LIN {X 0,Y 388.973,Z 474.655,A -85,B 0,C 180,E1 -11902.254,E2 -11902.254} C_VEL
LIN {X 0,Y 390.4,Z 456.308,A -85,B 0,C 180,E1 -11905.598,E2 -11905.598} C_VEL
LIN {X 0,Y 390.366,Z 451.941,A -85,B 0,C 180,E1 -11906.461,E2 -11906.461} C_VEL
LIN {X 0,Y 388.692,Z 443.592,A -85,B 0,C 180,E1 -11908.299,E2 -11908.299} C_VEL
LIN {X 0,Y 386.693,Z 436.556,A -85,B 0,C 180,E1 -11909.986,E2 -11909.986} C_VEL
LIN {X 0,Y 383.976,Z 428.562,A -85,B 0,C 180,E1 -11912.059,E2 -11912.059} C_VEL
LIN {X 0,Y 383.014,Z 425.779,A -85,B 0,C 180,E1 -11912.861,E2 -11912.861} C_VEL
LIN {X 0,Y 383.034,Z 425.772,A -85,B 0,C 180,E1 -11916.164,E2 -11916.164} C_VEL
LIN {X 0,Y 383.01,Z 425.774,A -85,B 0,C 180,E1 -11919.958,E2 -11919.958} C_VEL
LIN {X 0,Y 383.007,Z 425.776,A -85,B 0,C 180,E1 -11922.779,E2 -11922.779} C_VEL
LIN {X 0,Y 382.999,Z 425.778,A -85,B 0,C 180,E1 -11925.789,E2 -11925.789} C_VEL
LIN {X 0,Y 382.99,Z 425.776,A -85,B 0,C 180,E1 -11928.796,E2 -11928.796} C_VEL
LIN {X 0,Y 383.001,Z 425.776,A -85,B 0,C 180,E1 -11932.096,E2 -11932.096} C_VEL
LIN {X 0,Y 383.02,Z 425.775,A -85,B 0,C 180,E1 -11935.332,E2 -11935.332} C_VEL
LIN {X 0,Y 383.022,Z 425.882,A -85,B 0,C 180,E1 -11938.509,E2 -11938.509} C_VEL
LIN {X 0,Y 386.811,Z 443.638,A -85,B 0,C 180,E1 -11942.071,E2 -11942.071} C_VEL
LIN {X 0,Y 387.334,Z 447.211,A -85,B 0,C 180,E1 -11942.759,E2 -11942.759} C_VEL
LIN {X 0,Y 386.152,Z 463.005,A -85,B 0,C 180,E1 -11945.62,E2 -11945.62} C_VEL
LIN {X 0,Y 385.72,Z 469.471,A -85,B 0,C 180,E1 -11946.76,E2 -11946.76} C_VEL
LIN {X 0,Y 387.23,Z 483.824,A -85,B 0,C 180,E1 -11947.858,E2 -11947.858} C_VEL
LIN {X 0,Y 389.694,Z 500.187,A -85,B 0,C 180,E1 -11948.651,E2 -11948.651} C_VEL
LIN {X 0,Y 391.644,Z 523.161,A -85,B 0,C 180,E1 -11949.556,E2 -11949.556} C_VEL
LIN {X 0,Y 388.702,Z 598.961,A -85,B 0,C 180,E1 -11951.588,E2 -11951.588} C_VEL
LIN {X 0,Y 388.096,Z 612.843,A -85,B 0,C 180,E1 -11952.036,E2 -11952.036} C_VEL
LIN {X 0,Y 387.433,Z 625.993,A -85,B 0,C 180,E1 -11952.652,E2 -11952.652} C_VEL
LIN {X 0,Y 386.462,Z 638.87,A -85,B 0,C 180,E1 -11953.492,E2 -11953.492} C_VEL
LIN {X 0,Y 385.655,Z 649.554,A -85,B 0,C 180,E1 -11954.407,E2 -11954.407} C_VEL
LIN {X 0,Y 384.808,Z 660.326,A -85,B 0,C 180,E1 -11955.578,E2 -11955.578} C_VEL
LIN {X 0,Y 383.983,Z 669.284,A -85,B 0,C 180,E1 -11956.774,E2 -11956.774} C_VEL
LIN {X 0,Y 383.117,Z 678.923,A -85,B 0,C 180,E1 -11958.358,E2 -11958.358} C_VEL
LIN {X 0,Y 382.509,Z 686.731,A -85,B 0,C 180,E1 -11959.948,E2 -11959.948} C_VEL
LIN {X 0,Y 382.085,Z 692.947,A -85,B 0,C 180,E1 -11961.538,E2 -11961.538} C_VEL
LIN {X 0,Y 381.834,Z 697.818,A -85,B 0,C 180,E1 -11963.129,E2 -11963.129} C_VEL
LIN {X 0,Y 381.699,Z 701.49,A -85,B 0,C 180,E1 -11964.718,E2 -11964.718} C_VEL
LIN {X 0,Y 381.686,Z 703.304,A -85,B 0,C 180,E1 -11965.776,E2 -11965.776} C_VEL
LIN {X 0,Y 381.62,Z 704.68,A -85,B 0,C 180,E1 -11966.833,E2 -11966.833} C_VEL
LIN {X 0,Y 381.631,Z 705.587,A -85,B 0,C 180,E1 -11967.889,E2 -11967.889} C_VEL
LIN {X 0,Y 381.687,Z 706.203,A -85,B 0,C 180,E1 -11970,E2 -11970} C_VEL
LIN {X 0,Y 381.677,Z 705.98,A -85,B 0,C 180,E1 -11971.055,E2 -11971.055} C_VEL
LIN {X 0,Y 381.636,Z 705.361,A -85,B 0,C 180,E1 -11972.111,E2 -11972.111} C_VEL
LIN {X 0,Y 381.625,Z 704.35,A -85,B 0,C 180,E1 -11973.167,E2 -11973.167} C_VEL
LIN {X 0,Y 381.69,Z 702.918,A -85,B 0,C 180,E1 -11974.224,E2 -11974.224} C_VEL
LIN {X 0,Y 381.756,Z 698.991,A -85,B 0,C 180,E1 -11976.213,E2 -11976.213} C_VEL
LIN {X 0,Y 381.995,Z 694.268,A -85,B 0,C 180,E1 -11977.931,E2 -11977.931} C_VEL
LIN {X 0,Y 382.45,Z 687.532,A -85,B 0,C 180,E1 -11979.787,E2 -11979.787} C_VEL
LIN {X 0,Y 383.006,Z 680.171,A -85,B 0,C 180,E1 -11981.377,E2 -11981.377} C_VEL
LIN {X 0,Y 383.706,Z 672.652,A -85,B 0,C 180,E1 -11982.697,E2 -11982.697} C_VEL
LIN {X 0,Y 384.542,Z 663.035,A -85,B 0,C 180,E1 -11984.079,E2 -11984.079} C_VEL
LIN {X 0,Y 385.394,Z 652.076,A -85,B 0,C 180,E1 -11985.333,E2 -11985.333} C_VEL
LIN {X 0,Y 386.372,Z 640.484,A -85,B 0,C 180,E1 -11986.376,E2 -11986.376} C_VEL
LIN {X 0,Y 387.296,Z 628.071,A -85,B 0,C 180,E1 -11987.218,E2 -11987.218} C_VEL
LIN {X 0,Y 388.001,Z 614.983,A -85,B 0,C 180,E1 -11987.866,E2 -11987.866} C_VEL
LIN {X 0,Y 389.326,Z 594.994,A -85,B 0,C 180,E1 -11988.722,E2 -11988.722} C_VEL
LIN {X 0,Y 390.088,Z 575.45,A -85,B 0,C 180,E1 -11989.264,E2 -11989.264} C_VEL
LIN {X 0,Y 391.896,Z 521.918,A -85,B 0,C 180,E1 -11990.668,E2 -11990.668} C_VEL
LIN {X 0,Y 390.385,Z 503.692,A -85,B 0,C 180,E1 -11991.348,E2 -11991.348} C_VEL
LIN {X 0,Y 387.383,Z 484.338,A -85,B 0,C 180,E1 -11992.23,E2 -11992.23} C_VEL
LIN {X 0,Y 386.082,Z 477.709,A -85,B 0,C 180,E1 -11992.58,E2 -11992.58} C_VEL
LIN {X 0,Y 387.967,Z 460.117,A -85,B 0,C 180,E1 -11996.059,E2 -11996.059} C_VEL
LIN {X 0,Y 389.025,Z 450.691,A -85,B 0,C 180,E1 -11998.015,E2 -11998.015} C_VEL
LIN {X 0,Y 387.628,Z 442.996,A -85,B 0,C 180,E1 -11999.932,E2 -11999.932} C_VEL
LIN {X 0,Y 385.295,Z 433.56,A -85,B 0,C 180,E1 -12002.584,E2 -12002.584} C_VEL
LIN {X 0,Y 383.068,Z 425.77,A -85,B 0,C 180,E1 -12005.144,E2 -12005.144} C_VEL
LIN {X 0,Y 383.003,Z 425.777,A -85,B 0,C 180,E1 -12008.601,E2 -12008.601} C_VEL
LIN {X 0,Y 382.983,Z 425.78,A -85,B 0,C 180,E1 -12011.348,E2 -12011.348} C_VEL
LIN {X 0,Y 382.997,Z 425.778,A -85,B 0,C 180,E1 -12014.303,E2 -12014.303} C_VEL
LIN {X 0,Y 383.012,Z 425.777,A -85,B 0,C 180,E1 -12017.24,E2 -12017.24} C_VEL
LIN {X 0,Y 383.017,Z 425.775,A -85,B 0,C 180,E1 -12020.413,E2 -12020.413} C_VEL
LIN {X 0,Y 383.027,Z 425.772,A -85,B 0,C 180,E1 -12024.045,E2 -12024.045} C_VEL
LIN {X 0,Y 382.989,Z 425.778,A -85,B 0,C 180,E1 -12027.578,E2 -12027.578} C_VEL
LIN {X 0,Y 382.994,Z 425.778,A -85,B 0,C 180,E1 -12030.3,E2 -12030.3} C_VEL
LIN {X 0,Y 383.082,Z 425.769,A -85,B 0,C 180,E1 -12034.021,E2 -12034.021} C_VEL
LIN {X 0,Y 383.06,Z 425.881,A -85,B 0,C 180,E1 -12037.093,E2 -12037.093} C_VEL
LIN {X 0,Y 383.156,Z 426.461,A -85,B 0,C 180,E1 -12037.246,E2 -12037.246} C_VEL
LIN {X 0,Y 384.382,Z 429.177,A -85,B 0,C 180,E1 -12037.475,E2 -12037.475} C_VEL
LIN {X 0,Y 385.896,Z 431.761,A -85,B 0,C 180,E1 -12037.727,E2 -12037.727} C_VEL
LIN {X 0,Y 391.372,Z 442.113,A -85,B 0,C 180,E1 -12038.631,E2 -12038.631} C_VEL
LIN {X 0,Y 394.03,Z 448.2,A -85,B 0,C 180,E1 -12039.076,E2 -12039.076} C_VEL
LIN {X 0,Y 391.15,Z 515.753,A -85,B 0,C 180,E1 -12040.892,E2 -12040.892} C_VEL
LIN {X 0,Y 390.648,Z 532.946,A -85,B 0,C 180,E1 -12041.411,E2 -12041.411} C_VEL
LIN {X 0,Y 390.136,Z 545.919,A -85,B 0,C 180,E1 -12042.031,E2 -12042.031} C_VEL
LIN {X 0,Y 389.456,Z 558.538,A -85,B 0,C 180,E1 -12042.853,E2 -12042.853} C_VEL
LIN {X 0,Y 388.498,Z 570.752,A -85,B 0,C 180,E1 -12043.891,E2 -12043.891} C_VEL
LIN {X 0,Y 387.531,Z 581.387,A -85,B 0,C 180,E1 -12045.023,E2 -12045.023} C_VEL
LIN {X 0,Y 386.635,Z 591.162,A -85,B 0,C 180,E1 -12046.331,E2 -12046.331} C_VEL
LIN {X 0,Y 385.652,Z 600.607,A -85,B 0,C 180,E1 -12047.903,E2 -12047.903} C_VEL
LIN {X 0,Y 384.683,Z 608.126,A -85,B 0,C 180,E1 -12049.473,E2 -12049.473} C_VEL
LIN {X 0,Y 383.999,Z 614.699,A -85,B 0,C 180,E1 -12051.235,E2 -12051.235} C_VEL
LIN {X 0,Y 383.308,Z 618.819,A -85,B 0,C 180,E1 -12052.626,E2 -12052.626} C_VEL
LIN {X 0,Y 383.106,Z 621.312,A -85,B 0,C 180,E1 -12053.681,E2 -12053.681} C_VEL
LIN {X 0,Y 382.945,Z 623.281,A -85,B 0,C 180,E1 -12054.735,E2 -12054.735} C_VEL
LIN {X 0,Y 382.672,Z 624.822,A -85,B 0,C 180,E1 -12055.787,E2 -12055.787} C_VEL
LIN {X 0,Y 382.364,Z 625.951,A -85,B 0,C 180,E1 -12056.839,E2 -12056.839} C_VEL
LIN {X 0,Y 382.146,Z 626.62,A -85,B 0,C 180,E1 -12057.892,E2 -12057.892} C_VEL
LIN {X 0,Y 382.038,Z 626.843,A -85,B 0,C 180,E1 -12058.946,E2 -12058.946} C_VEL
LIN {X 0,Y 381.995,Z 626.656,A -85,B 0,C 180,E1 -12060,E2 -12060} C_VEL
LIN {X 0,Y 382.015,Z 626.047,A -85,B 0,C 180,E1 -12061.054,E2 -12061.054} C_VEL
LIN {X 0,Y 382.127,Z 624.97,A -85,B 0,C 180,E1 -12062.108,E2 -12062.108} C_VEL
LIN {X 0,Y 382.257,Z 623.479,A -85,B 0,C 180,E1 -12063.162,E2 -12063.162} C_VEL
LIN {X 0,Y 382.481,Z 620.399,A -85,B 0,C 180,E1 -12064.743,E2 -12064.743} C_VEL
LIN {X 0,Y 382.545,Z 616.243,A -85,B 0,C 180,E1 -12066.329,E2 -12066.329} C_VEL
LIN {X 0,Y 382.918,Z 609.948,A -85,B 0,C 180,E1 -12068.151,E2 -12068.151} C_VEL
LIN {X 0,Y 383.35,Z 602.81,A -85,B 0,C 180,E1 -12069.764,E2 -12069.764} C_VEL
LIN {X 0,Y 383.91,Z 594.085,A -85,B 0,C 180,E1 -12071.35,E2 -12071.35} C_VEL
LIN {X 0,Y 384.536,Z 584.075,A -85,B 0,C 180,E1 -12072.803,E2 -12072.803} C_VEL
LIN {X 0,Y 385.148,Z 574.024,A -85,B 0,C 180,E1 -12073.992,E2 -12073.992} C_VEL
LIN {X 0,Y 385.81,Z 562.335,A -85,B 0,C 180,E1 -12075.102,E2 -12075.102} C_VEL
LIN {X 0,Y 386.243,Z 550.748,A -85,B 0,C 180,E1 -12075.975,E2 -12075.975} C_VEL
LIN {X 0,Y 386.751,Z 538.186,A -85,B 0,C 180,E1 -12076.699,E2 -12076.699} C_VEL
LIN {X 0,Y 387.148,Z 525.23,A -85,B 0,C 180,E1 -12077.225,E2 -12077.225} C_VEL
LIN {X 0,Y 387.449,Z 505.59,A -85,B 0,C 180,E1 -12077.722,E2 -12077.722} C_VEL
LIN {X 0,Y 388.686,Z 442.712,A -85,B 0,C 180,E1 -12079.186,E2 -12079.186} C_VEL
LIN {X 0,Y 383.073,Z 425.774,A -85,B 0,C 180,E1 -12079.854,E2 -12079.854} C_VEL
LIN {X 0,Y 383.024,Z 425.771,A -85,B 0,C 180,E1 -12083.808,E2 -12083.808} C_VEL
LIN {X 0,Y 383.082,Z 425.764,A -85,B 0,C 180,E1 -12086.123,E2 -12086.123} C_VEL
LIN {X 0,Y 382.995,Z 425.777,A -85,B 0,C 180,E1 -12089.7,E2 -12089.7} C_VEL
LIN {X 0,Y 383.006,Z 425.755,A -85,B 0,C 180,E1 -12093.401,E2 -12093.401} C_VEL
LIN {X 0,Y 383.034,Z 425.77,A -85,B 0,C 180,E1 -12096.165,E2 -12096.165} C_VEL
LIN {X 0,Y 383.01,Z 425.764,A -85,B 0,C 180,E1 -12099.958,E2 -12099.958} C_VEL
LIN {X 0,Y 383.007,Z 425.778,A -85,B 0,C 180,E1 -12102.779,E2 -12102.779} C_VEL
LIN {X 0,Y 382.999,Z 425.763,A -85,B 0,C 180,E1 -12105.789,E2 -12105.789} C_VEL
LIN {X 0,Y 382.991,Z 425.775,A -85,B 0,C 180,E1 -12108.796,E2 -12108.796} C_VEL
LIN {X 0,Y 383.001,Z 425.778,A -85,B 0,C 180,E1 -12112.097,E2 -12112.097} C_VEL
LIN {X 0,Y 383.02,Z 425.773,A -85,B 0,C 180,E1 -12115.332,E2 -12115.332} C_VEL
LIN {X 0,Y 382.984,Z 425.783,A -85,B 0,C 180,E1 -12119.081,E2 -12119.081} C_VEL
LIN {X 0,Y 383.042,Z 425.845,A -85,B 0,C 180,E1 -12120.607,E2 -12120.607} C_VEL
LIN {X 0,Y 386.37,Z 440.616,A -85,B 0,C 180,E1 -12123.643,E2 -12123.643} C_VEL
LIN {X 0,Y 387.42,Z 446.111,A -85,B 0,C 180,E1 -12124.738,E2 -12124.738} C_VEL
LIN {X 0,Y 386.957,Z 457.171,A -85,B 0,C 180,E1 -12126.732,E2 -12126.732} C_VEL
LIN {X 0,Y 386.301,Z 472.125,A -85,B 0,C 180,E1 -12129.272,E2 -12129.272} C_VEL
LIN {X 0,Y 390.407,Z 495.726,A -85,B 0,C 180,E1 -12129.965,E2 -12129.965} C_VEL
LIN {X 0,Y 389.277,Z 577.449,A -85,B 0,C 180,E1 -12131.48,E2 -12131.48} C_VEL
LIN {X 0,Y 388.907,Z 590.427,A -85,B 0,C 180,E1 -12131.837,E2 -12131.837} C_VEL
LIN {X 0,Y 388.248,Z 603.511,A -85,B 0,C 180,E1 -12132.418,E2 -12132.418} C_VEL
LIN {X 0,Y 387.533,Z 615.074,A -85,B 0,C 180,E1 -12133.132,E2 -12133.132} C_VEL
LIN {X 0,Y 386.746,Z 626.393,A -85,B 0,C 180,E1 -12134.047,E2 -12134.047} C_VEL
LIN {X 0,Y 385.986,Z 636.548,A -85,B 0,C 180,E1 -12135.089,E2 -12135.089} C_VEL
LIN {X 0,Y 385.085,Z 645.997,A -85,B 0,C 180,E1 -12136.275,E2 -12136.275} C_VEL
LIN {X 0,Y 384.159,Z 654.573,A -85,B 0,C 180,E1 -12137.587,E2 -12137.587} C_VEL
LIN {X 0,Y 383.435,Z 662.923,A -85,B 0,C 180,E1 -12139.171,E2 -12139.171} C_VEL
LIN {X 0,Y 382.866,Z 668.604,A -85,B 0,C 180,E1 -12140.491,E2 -12140.491} C_VEL
LIN {X 0,Y 382.345,Z 674.129,A -85,B 0,C 180,E1 -12142.076,E2 -12142.076} C_VEL
LIN {X 0,Y 382.158,Z 677.456,A -85,B 0,C 180,E1 -12143.259,E2 -12143.259} C_VEL
LIN {X 0,Y 381.297,Z 679.476,A -85,B 0,C 180,E1 -12144.086,E2 -12144.086} C_VEL
LIN {X 0,Y 378.194,Z 682.226,A -85,B 0,C 180,E1 -12145.446,E2 -12145.446} C_VEL
LIN {X 0,Y 375.209,Z 684.278,A -85,B 0,C 180,E1 -12146.854,E2 -12146.854} C_VEL
LIN {X 0,Y 374.545,Z 685.111,A -85,B 0,C 180,E1 -12147.741,E2 -12147.741} C_VEL
LIN {X 0,Y 374.545,Z 685.825,A -85,B 0,C 180,E1 -12148.925,E2 -12148.925} C_VEL
LIN {X 0,Y 374.538,Z 686.06,A -85,B 0,C 180,E1 -12150,E2 -12150} C_VEL
LIN {X 0,Y 374.545,Z 685.868,A -85,B 0,C 180,E1 -12151.075,E2 -12151.075} C_VEL
LIN {X 0,Y 374.566,Z 684.317,A -85,B 0,C 180,E1 -12153.227,E2 -12153.227} C_VEL
LIN {X 0,Y 374.669,Z 682.951,A -85,B 0,C 180,E1 -12154.303,E2 -12154.303} C_VEL
LIN {X 0,Y 374.925,Z 680.078,A -85,B 0,C 180,E1 -12155.918,E2 -12155.918} C_VEL
LIN {X 0,Y 375.16,Z 676.178,A -85,B 0,C 180,E1 -12157.535,E2 -12157.535} C_VEL
LIN {X 0,Y 375.63,Z 671.12,A -85,B 0,C 180,E1 -12159.151,E2 -12159.151} C_VEL
LIN {X 0,Y 376.267,Z 664.744,A -85,B 0,C 180,E1 -12160.765,E2 -12160.765} C_VEL
LIN {X 0,Y 377.057,Z 656.821,A -85,B 0,C 180,E1 -12162.377,E2 -12162.377} C_VEL
LIN {X 0,Y 377.991,Z 648.72,A -85,B 0,C 180,E1 -12163.713,E2 -12163.713} C_VEL
LIN {X 0,Y 378.941,Z 638.763,A -85,B 0,C 180,E1 -12165.049,E2 -12165.049} C_VEL
LIN {X 0,Y 379.824,Z 627.571,A -85,B 0,C 180,E1 -12166.252,E2 -12166.252} C_VEL
LIN {X 0,Y 380.683,Z 616.598,A -85,B 0,C 180,E1 -12167.181,E2 -12167.181} C_VEL
LIN {X 0,Y 381.51,Z 605.445,A -85,B 0,C 180,E1 -12167.903,E2 -12167.903} C_VEL
LIN {X 0,Y 382.133,Z 592.169,A -85,B 0,C 180,E1 -12168.532,E2 -12168.532} C_VEL
LIN {X 0,Y 382.513,Z 580.383,A -85,B 0,C 180,E1 -12168.895,E2 -12168.895} C_VEL
LIN {X 0,Y 383.723,Z 496.111,A -85,B 0,C 180,E1 -12170.494,E2 -12170.494} C_VEL
LIN {X 0,Y 379.532,Z 472.111,A -85,B 0,C 180,E1 -12171.239,E2 -12171.239} C_VEL
LIN {X 0,Y 380.142,Z 457.818,A -85,B 0,C 180,E1 -12173.71,E2 -12173.71} C_VEL
LIN {X 0,Y 380.63,Z 448.418,A -85,B 0,C 180,E1 -12175.393,E2 -12175.393} C_VEL
LIN {X 0,Y 378.451,Z 437.346,A -85,B 0,C 180,E1 -12177.663,E2 -12177.663} C_VEL
LIN {X 0,Y 375.968,Z 426.654,A -85,B 0,C 180,E1 -12179.926,E2 -12179.926} C_VEL
LIN {X 0,Y 375.951,Z 426.657,A -85,B 0,C 180,E1 -12182.828,E2 -12182.828} C_VEL
LIN {X 0,Y 375.959,Z 426.656,A -85,B 0,C 180,E1 -12185.415,E2 -12185.415} C_VEL
LIN {X 0,Y 375.975,Z 426.651,A -85,B 0,C 180,E1 -12188.27,E2 -12188.27} C_VEL
LIN {X 0,Y 375.937,Z 426.659,A -85,B 0,C 180,E1 -12191.601,E2 -12191.601} C_VEL
LIN {X 0,Y 375.957,Z 426.658,A -85,B 0,C 180,E1 -12195.264,E2 -12195.264} C_VEL
LIN {X 0,Y 375.943,Z 426.652,A -85,B 0,C 180,E1 -12199.133,E2 -12199.133} C_VEL
LIN {X 0,Y 375.966,Z 426.651,A -85,B 0,C 180,E1 -12201.912,E2 -12201.912} C_VEL
LIN {X 0,Y 375.982,Z 426.649,A -85,B 0,C 180,E1 -12205.333,E2 -12205.333} C_VEL
LIN {X 0,Y 375.96,Z 426.656,A -85,B 0,C 180,E1 -12208.438,E2 -12208.438} C_VEL
LIN {X 0,Y 376.019,Z 426.689,A -85,B 0,C 180,E1 -12211.117,E2 -12211.117} C_VEL
LIN {X 0,Y 379.558,Z 443.932,A -85,B 0,C 180,E1 -12214.5,E2 -12214.5} C_VEL
LIN {X 0,Y 379.934,Z 447.448,A -85,B 0,C 180,E1 -12215.17,E2 -12215.17} C_VEL
LIN {X 0,Y 379.113,Z 462.901,A -85,B 0,C 180,E1 -12217.957,E2 -12217.957} C_VEL
LIN {X 0,Y 378.643,Z 472.829,A -85,B 0,C 180,E1 -12219.74,E2 -12219.74} C_VEL
LIN {X 0,Y 381.87,Z 496.426,A -85,B 0,C 180,E1 -12220.465,E2 -12220.465} C_VEL
LIN {X 0,Y 379.956,Z 584.101,A -85,B 0,C 180,E1 -12222.577,E2 -12222.577} C_VEL
LIN {X 0,Y 379.453,Z 597.319,A -85,B 0,C 180,E1 -12223.109,E2 -12223.109} C_VEL
LIN {X 0,Y 378.89,Z 610.179,A -85,B 0,C 180,E1 -12223.845,E2 -12223.845} C_VEL
LIN {X 0,Y 378.172,Z 622.529,A -85,B 0,C 180,E1 -12224.781,E2 -12224.781} C_VEL
LIN {X 0,Y 377.587,Z 633.478,A -85,B 0,C 180,E1 -12225.839,E2 -12225.839} C_VEL
LIN {X 0,Y 376.872,Z 643.781,A -85,B 0,C 180,E1 -12227.069,E2 -12227.069} C_VEL
LIN {X 0,Y 376.221,Z 653.014,A -85,B 0,C 180,E1 -12228.415,E2 -12228.415} C_VEL
LIN {X 0,Y 375.622,Z 661.929,A -85,B 0,C 180,E1 -12230.034,E2 -12230.034} C_VEL
LIN {X 0,Y 375.143,Z 669.112,A -85,B 0,C 180,E1 -12231.652,E2 -12231.652} C_VEL
LIN {X 0,Y 374.831,Z 675.609,A -85,B 0,C 180,E1 -12233.541,E2 -12233.541} C_VEL
LIN {X 0,Y 374.708,Z 679.841,A -85,B 0,C 180,E1 -12235.158,E2 -12235.158} C_VEL
LIN {X 0,Y 374.529,Z 682.942,A -85,B 0,C 180,E1 -12236.773,E2 -12236.773} C_VEL
LIN {X 0,Y 374.518,Z 684.403,A -85,B 0,C 180,E1 -12237.849,E2 -12237.849} C_VEL
LIN {X 0,Y 374.511,Z 685.432,A -85,B 0,C 180,E1 -12238.925,E2 -12238.925} C_VEL
LIN {X 0,Y 374.538,Z 686.048,A -85,B 0,C 180,E1 -12240,E2 -12240} C_VEL
LIN {X 0,Y 374.563,Z 686.185,A -85,B 0,C 180,E1 -12241.075,E2 -12241.075} C_VEL
LIN {X 0,Y 374.606,Z 685.905,A -85,B 0,C 180,E1 -12242.15,E2 -12242.15} C_VEL
LIN {X 0,Y 374.62,Z 685.213,A -85,B 0,C 180,E1 -12243.226,E2 -12243.226} C_VEL
LIN {X 0,Y 374.676,Z 684.042,A -85,B 0,C 180,E1 -12244.303,E2 -12244.303} C_VEL
LIN {X 0,Y 375.059,Z 681.456,A -85,B 0,C 180,E1 -12245.915,E2 -12245.915} C_VEL
LIN {X 0,Y 375.265,Z 677.811,A -85,B 0,C 180,E1 -12247.533,E2 -12247.533} C_VEL
LIN {X 0,Y 375.795,Z 672.997,A -85,B 0,C 180,E1 -12249.147,E2 -12249.147} C_VEL
LIN {X 0,Y 376.446,Z 666.921,A -85,B 0,C 180,E1 -12250.76,E2 -12250.76} C_VEL
LIN {X 0,Y 377.356,Z 659.254,A -85,B 0,C 180,E1 -12252.367,E2 -12252.367} C_VEL
LIN {X 0,Y 378.294,Z 649.736,A -85,B 0,C 180,E1 -12253.976,E2 -12253.976} C_VEL
LIN {X 0,Y 379.544,Z 638.677,A -85,B 0,C 180,E1 -12255.443,E2 -12255.443} C_VEL
LIN {X 0,Y 380.63,Z 627.513,A -85,B 0,C 180,E1 -12256.63,E2 -12256.63} C_VEL
LIN {X 0,Y 381.746,Z 614.971,A -85,B 0,C 180,E1 -12257.684,E2 -12257.684} C_VEL
LIN {X 0,Y 382.649,Z 602.665,A -85,B 0,C 180,E1 -12258.471,E2 -12258.471} C_VEL
LIN {X 0,Y 383.412,Z 589.501,A -85,B 0,C 180,E1 -12259.092,E2 -12259.092} C_VEL
LIN {X 0,Y 384.174,Z 573.253,A -85,B 0,C 180,E1 -12259.573,E2 -12259.573} C_VEL
LIN {X 0,Y 387.33,Z 497.701,A -85,B 0,C 180,E1 -12261.645,E2 -12261.645} C_VEL
LIN {X 0,Y 384.771,Z 483.743,A -85,B 0,C 180,E1 -12262.36,E2 -12262.36} C_VEL
LIN {X 0,Y 382.635,Z 474.89,A -85,B 0,C 180,E1 -12262.905,E2 -12262.905} C_VEL
LIN {X 0,Y 384.128,Z 457.935,A -85,B 0,C 180,E1 -12266.047,E2 -12266.047} C_VEL
LIN {X 0,Y 383.857,Z 453.55,A -85,B 0,C 180,E1 -12266.945,E2 -12266.945} C_VEL
LIN {X 0,Y 381.9,Z 444.492,A -85,B 0,C 180,E1 -12269.05,E2 -12269.05} C_VEL
LIN {X 0,Y 379.337,Z 435.98,A -85,B 0,C 180,E1 -12271.249,E2 -12271.249} C_VEL
LIN {X 0,Y 377.124,Z 429.72,A -85,B 0,C 180,E1 -12273.006,E2 -12273.006} C_VEL
LIN {X 0,Y 375.977,Z 426.653,A -85,B 0,C 180,E1 -12273.948,E2 -12273.948} C_VEL
LIN {X 0,Y 375.955,Z 426.654,A -85,B 0,C 180,E1 -12276.741,E2 -12276.741} C_VEL
LIN {X 0,Y 375.99,Z 426.648,A -85,B 0,C 180,E1 -12279.971,E2 -12279.971} C_VEL
LIN {X 0,Y 375.932,Z 426.657,A -85,B 0,C 180,E1 -12283.766,E2 -12283.766} C_VEL
LIN {X 0,Y 375.936,Z 426.655,A -85,B 0,C 180,E1 -12286.811,E2 -12286.811} C_VEL
LIN {X 0,Y 375.964,Z 426.651,A -85,B 0,C 180,E1 -12290.537,E2 -12290.537} C_VEL
LIN {X 0,Y 375.965,Z 426.653,A -85,B 0,C 180,E1 -12293.496,E2 -12293.496} C_VEL
LIN {X 0,Y 375.962,Z 426.652,A -85,B 0,C 180,E1 -12295.889,E2 -12295.889} C_VEL
LIN {X 0,Y 375.984,Z 426.784,A -85,B 0,C 180,E1 -12298.283,E2 -12298.283} C_VEL
LIN {X 0,Y 379.69,Z 444.183,A -85,B 0,C 180,E1 -12301.836,E2 -12301.836} C_VEL
LIN {X 0,Y 380.366,Z 449.085,A -85,B 0,C 180,E1 -12302.796,E2 -12302.796} C_VEL
LIN {X 0,Y 379.119,Z 464.66,A -85,B 0,C 180,E1 -12305.621,E2 -12305.621} C_VEL
LIN {X 0,Y 380.633,Z 479.637,A -85,B 0,C 180,E1 -12306.898,E2 -12306.898} C_VEL
LIN {X 0,Y 381.331,Z 485.609,A -85,B 0,C 180,E1 -12307.328,E2 -12307.328} C_VEL
LIN {X 0,Y 383.696,Z 501.63,A -85,B 0,C 180,E1 -12308.134,E2 -12308.134} C_VEL
LIN {X 0,Y 385.511,Z 524.207,A -85,B 0,C 180,E1 -12309.054,E2 -12309.054} C_VEL
LIN {X 0,Y 382.542,Z 594.05,A -85,B 0,C 180,E1 -12311.002,E2 -12311.002} C_VEL
LIN {X 0,Y 381.798,Z 610.283,A -85,B 0,C 180,E1 -12311.486,E2 -12311.486} C_VEL
LIN {X 0,Y 380.957,Z 624.045,A -85,B 0,C 180,E1 -12312.139,E2 -12312.139} C_VEL
LIN {X 0,Y 380.017,Z 636.183,A -85,B 0,C 180,E1 -12312.927,E2 -12312.927} C_VEL
LIN {X 0,Y 378.963,Z 648.609,A -85,B 0,C 180,E1 -12313.987,E2 -12313.987} C_VEL
LIN {X 0,Y 378.074,Z 659.411,A -85,B 0,C 180,E1 -12315.156,E2 -12315.156} C_VEL
LIN {X 0,Y 377.093,Z 669.669,A -85,B 0,C 180,E1 -12316.528,E2 -12316.528} C_VEL
LIN {X 0,Y 376.34,Z 677.825,A -85,B 0,C 180,E1 -12317.872,E2 -12317.872} C_VEL
LIN {X 0,Y 375.596,Z 685.767,A -85,B 0,C 180,E1 -12319.488,E2 -12319.488} C_VEL
LIN {X 0,Y 375.191,Z 691.184,A -85,B 0,C 180,E1 -12320.838,E2 -12320.838} C_VEL
LIN {X 0,Y 374.819,Z 696.396,A -85,B 0,C 180,E1 -12322.458,E2 -12322.458} C_VEL
LIN {X 0,Y 374.662,Z 699.837,A -85,B 0,C 180,E1 -12323.821,E2 -12323.821} C_VEL
LIN {X 0,Y 374.609,Z 703.242,A -85,B 0,C 180,E1 -12325.696,E2 -12325.696} C_VEL
LIN {X 0,Y 374.531,Z 704.583,A -85,B 0,C 180,E1 -12326.773,E2 -12326.773} C_VEL
LIN {X 0,Y 374.529,Z 705.43,A -85,B 0,C 180,E1 -12327.849,E2 -12327.849} C_VEL
LIN {X 0,Y 374.618,Z 706.015,A -85,B 0,C 180,E1 -12330,E2 -12330} C_VEL
LIN {X 0,Y 374.577,Z 705.791,A -85,B 0,C 180,E1 -12331.075,E2 -12331.075} C_VEL
LIN {X 0,Y 374.536,Z 704.161,A -85,B 0,C 180,E1 -12333.227,E2 -12333.227} C_VEL
LIN {X 0,Y 374.611,Z 702.728,A -85,B 0,C 180,E1 -12334.304,E2 -12334.304} C_VEL
LIN {X 0,Y 374.678,Z 699.099,A -85,B 0,C 180,E1 -12336.202,E2 -12336.202} C_VEL
LIN {X 0,Y 374.923,Z 694.078,A -85,B 0,C 180,E1 -12338.082,E2 -12338.082} C_VEL
LIN {X 0,Y 375.335,Z 688.439,A -85,B 0,C 180,E1 -12339.702,E2 -12339.702} C_VEL
LIN {X 0,Y 375.89,Z 681.336,A -85,B 0,C 180,E1 -12341.322,E2 -12341.322} C_VEL
LIN {X 0,Y 376.749,Z 672.466,A -85,B 0,C 180,E1 -12342.935,E2 -12342.935} C_VEL
LIN {X 0,Y 377.562,Z 663.623,A -85,B 0,C 180,E1 -12344.24,E2 -12344.24} C_VEL
LIN {X 0,Y 378.432,Z 653.179,A -85,B 0,C 180,E1 -12345.484,E2 -12345.484} C_VEL
LIN {X 0,Y 379.419,Z 641.887,A -85,B 0,C 180,E1 -12346.546,E2 -12346.546} C_VEL
LIN {X 0,Y 380.364,Z 630.119,A -85,B 0,C 180,E1 -12347.403,E2 -12347.403} C_VEL
LIN {X 0,Y 381.092,Z 617.821,A -85,B 0,C 180,E1 -12348.062,E2 -12348.062} C_VEL
LIN {X 0,Y 382.627,Z 598.072,A -85,B 0,C 180,E1 -12349.028,E2 -12349.028} C_VEL
LIN {X 0,Y 383.412,Z 583.589,A -85,B 0,C 180,E1 -12349.509,E2 -12349.509} C_VEL
LIN {X 0,Y 385.674,Z 523.098,A -85,B 0,C 180,E1 -12351.137,E2 -12351.137} C_VEL
LIN {X 0,Y 384.099,Z 503.644,A -85,B 0,C 180,E1 -12351.897,E2 -12351.897} C_VEL
LIN {X 0,Y 381.181,Z 484.996,A -85,B 0,C 180,E1 -12352.798,E2 -12352.798} C_VEL
LIN {X 0,Y 379.49,Z 476.567,A -85,B 0,C 180,E1 -12353.276,E2 -12353.276} C_VEL
LIN {X 0,Y 381.779,Z 457.87,A -85,B 0,C 180,E1 -12357.104,E2 -12357.104} C_VEL
LIN {X 0,Y 382.287,Z 452.33,A -85,B 0,C 180,E1 -12358.317,E2 -12358.317} C_VEL
LIN {X 0,Y 380.977,Z 445.123,A -85,B 0,C 180,E1 -12360.178,E2 -12360.178} C_VEL
LIN {X 0,Y 378.656,Z 435.605,A -85,B 0,C 180,E1 -12362.964,E2 -12362.964} C_VEL
LIN {X 0,Y 376.585,Z 428.685,A -85,B 0,C 180,E1 -12365.348,E2 -12365.348} C_VEL
LIN {X 0,Y 376.009,Z 426.649,A -85,B 0,C 180,E1 -12366.177,E2 -12366.177} C_VEL
LIN {X 0,Y 375.989,Z 426.651,A -85,B 0,C 180,E1 -12369.97,E2 -12369.97} C_VEL
LIN {X 0,Y 375.931,Z 426.657,A -85,B 0,C 180,E1 -12373.766,E2 -12373.766} C_VEL
LIN {X 0,Y 375.936,Z 426.656,A -85,B 0,C 180,E1 -12376.811,E2 -12376.811} C_VEL
LIN {X 0,Y 375.965,Z 426.654,A -85,B 0,C 180,E1 -12380.538,E2 -12380.538} C_VEL
LIN {X 0,Y 375.966,Z 426.654,A -85,B 0,C 180,E1 -12383.496,E2 -12383.496} C_VEL
LIN {X 0,Y 375.962,Z 426.651,A -85,B 0,C 180,E1 -12385.889,E2 -12385.889} C_VEL
LIN {X 0,Y 375.967,Z 426.654,A -85,B 0,C 180,E1 -12389.688,E2 -12389.688} C_VEL
LIN {X 0,Y 376.022,Z 426.651,A -85,B 0,C 180,E1 -12393.348,E2 -12393.348} C_VEL
LIN {X 0,Y 376.008,Z 426.687,A -85,B 0,C 180,E1 -12396.087,E2 -12396.087} C_VEL
LIN {X 0,Y 376.203,Z 427.627,A -85,B 0,C 180,E1 -12396.478,E2 -12396.478} C_VEL
LIN {X 0,Y 377.551,Z 430.253,A -85,B 0,C 180,E1 -12396.74,E2 -12396.74} C_VEL
LIN {X 0,Y 382.796,Z 439.566,A -85,B 0,C 180,E1 -12397.672,E2 -12397.672} C_VEL
LIN {X 0,Y 387.808,Z 449.945,A -85,B 0,C 180,E1 -12398.555,E2 -12398.555} C_VEL
LIN {X 0,Y 384.941,Z 514.456,A -85,B 0,C 180,E1 -12400.364,E2 -12400.364} C_VEL
LIN {X 0,Y 384.336,Z 532.731,A -85,B 0,C 180,E1 -12400.921,E2 -12400.921} C_VEL
LIN {X 0,Y 383.828,Z 545.491,A -85,B 0,C 180,E1 -12401.519,E2 -12401.519} C_VEL
LIN {X 0,Y 383.077,Z 558.743,A -85,B 0,C 180,E1 -12402.38,E2 -12402.38} C_VEL
LIN {X 0,Y 382.112,Z 570.508,A -85,B 0,C 180,E1 -12403.377,E2 -12403.377} C_VEL
LIN {X 0,Y 380.977,Z 582.063,A -85,B 0,C 180,E1 -12404.622,E2 -12404.622} C_VEL
LIN {X 0,Y 380.085,Z 590.949,A -85,B 0,C 180,E1 -12405.818,E2 -12405.818} C_VEL
LIN {X 0,Y 379.017,Z 600.576,A -85,B 0,C 180,E1 -12407.416,E2 -12407.416} C_VEL
LIN {X 0,Y 378.037,Z 608.303,A -85,B 0,C 180,E1 -12409.015,E2 -12409.015} C_VEL
LIN {X 0,Y 377.269,Z 614.587,A -85,B 0,C 180,E1 -12410.68,E2 -12410.68} C_VEL
LIN {X 0,Y 376.374,Z 619.889,A -85,B 0,C 180,E1 -12412.489,E2 -12412.489} C_VEL
LIN {X 0,Y 376.139,Z 622.309,A -85,B 0,C 180,E1 -12413.563,E2 -12413.563} C_VEL
LIN {X 0,Y 375.938,Z 624.219,A -85,B 0,C 180,E1 -12414.637,E2 -12414.637} C_VEL
LIN {X 0,Y 375.651,Z 625.723,A -85,B 0,C 180,E1 -12415.708,E2 -12415.708} C_VEL
LIN {X 0,Y 375.332,Z 626.807,A -85,B 0,C 180,E1 -12416.78,E2 -12416.78} C_VEL
LIN {X 0,Y 375.103,Z 627.411,A -85,B 0,C 180,E1 -12417.853,E2 -12417.853} C_VEL
LIN {X 0,Y 374.986,Z 627.591,A -85,B 0,C 180,E1 -12418.926,E2 -12418.926} C_VEL
LIN {X 0,Y 374.941,Z 627.357,A -85,B 0,C 180,E1 -12420,E2 -12420} C_VEL
LIN {X 0,Y 374.965,Z 626.67,A -85,B 0,C 180,E1 -12421.074,E2 -12421.074} C_VEL
LIN {X 0,Y 375.083,Z 625.543,A -85,B 0,C 180,E1 -12422.148,E2 -12422.148} C_VEL
LIN {X 0,Y 375.194,Z 624.004,A -85,B 0,C 180,E1 -12423.221,E2 -12423.221} C_VEL
LIN {X 0,Y 375.431,Z 620.831,A -85,B 0,C 180,E1 -12424.832,E2 -12424.832} C_VEL
LIN {X 0,Y 375.514,Z 616.575,A -85,B 0,C 180,E1 -12426.448,E2 -12426.448} C_VEL
LIN {X 0,Y 375.877,Z 610.02,A -85,B 0,C 180,E1 -12428.332,E2 -12428.332} C_VEL
LIN {X 0,Y 376.336,Z 602.873,A -85,B 0,C 180,E1 -12429.947,E2 -12429.947} C_VEL
LIN {X 0,Y 376.816,Z 595.59,A -85,B 0,C 180,E1 -12431.294,E2 -12431.294} C_VEL
LIN {X 0,Y 377.43,Z 585.799,A -85,B 0,C 180,E1 -12432.775,E2 -12432.775} C_VEL
LIN {X 0,Y 378.124,Z 574.732,A -85,B 0,C 180,E1 -12434.12,E2 -12434.12} C_VEL
LIN {X 0,Y 378.827,Z 562.849,A -85,B 0,C 180,E1 -12435.267,E2 -12435.267} C_VEL
LIN {X 0,Y 379.252,Z 551.478,A -85,B 0,C 180,E1 -12436.139,E2 -12436.139} C_VEL
LIN {X 0,Y 379.789,Z 538.961,A -85,B 0,C 180,E1 -12436.876,E2 -12436.876} C_VEL
LIN {X 0,Y 380.21,Z 525.11,A -85,B 0,C 180,E1 -12437.445,E2 -12437.445} C_VEL
LIN {X 0,Y 380.636,Z 499.708,A -85,B 0,C 180,E1 -12438.085,E2 -12438.085} C_VEL
LIN {X 0,Y 381.856,Z 444.24,A -85,B 0,C 180,E1 -12439.41,E2 -12439.41} C_VEL
LIN {X 0,Y 376.035,Z 426.649,A -85,B 0,C 180,E1 -12440.122,E2 -12440.122} C_VEL
LIN {X 0,Y 375.989,Z 426.646,A -85,B 0,C 180,E1 -12444.282,E2 -12444.282} C_VEL
LIN {X 0,Y 376.022,Z 426.644,A -85,B 0,C 180,E1 -12446.652,E2 -12446.652} C_VEL
LIN {X 0,Y 375.967,Z 426.651,A -85,B 0,C 180,E1 -12450.313,E2 -12450.313} C_VEL
LIN {X 0,Y 375.962,Z 426.633,A -85,B 0,C 180,E1 -12454.111,E2 -12454.111} C_VEL
LIN {X 0,Y 375.956,Z 426.655,A -85,B 0,C 180,E1 -12456.741,E2 -12456.741} C_VEL
LIN {X 0,Y 375.99,Z 426.638,A -85,B 0,C 180,E1 -12459.971,E2 -12459.971} C_VEL
LIN {X 0,Y 375.932,Z 426.658,A -85,B 0,C 180,E1 -12463.766,E2 -12463.766} C_VEL
LIN {X 0,Y 375.936,Z 426.65,A -85,B 0,C 180,E1 -12466.811,E2 -12466.811} C_VEL
LIN {X 0,Y 375.964,Z 426.647,A -85,B 0,C 180,E1 -12470.537,E2 -12470.537} C_VEL
LIN {X 0,Y 375.966,Z 426.648,A -85,B 0,C 180,E1 -12473.496,E2 -12473.496} C_VEL
LIN {X 0,Y 375.962,Z 426.65,A -85,B 0,C 180,E1 -12475.889,E2 -12475.889} C_VEL
LIN {X 0,Y 375.966,Z 426.656,A -85,B 0,C 180,E1 -12479.687,E2 -12479.687} C_VEL
LIN {X 0,Y 375.98,Z 426.721,A -85,B 0,C 180,E1 -12480.23,E2 -12480.23} C_VEL
LIN {X 0,Y 379.182,Z 440.662,A -85,B 0,C 180,E1 -12483.149,E2 -12483.149} C_VEL
LIN {X 0,Y 380.629,Z 448.837,A -85,B 0,C 180,E1 -12484.789,E2 -12484.789} C_VEL
LIN {X 0,Y 379.708,Z 467.49,A -85,B 0,C 180,E1 -12488.093,E2 -12488.093} C_VEL
LIN {X 0,Y 379.49,Z 472.236,A -85,B 0,C 180,E1 -12488.88,E2 -12488.88} C_VEL
LIN {X 0,Y 383.754,Z 496.441,A -85,B 0,C 180,E1 -12489.614,E2 -12489.614} C_VEL
LIN {X 0,Y 382.422,Z 581.822,A -85,B 0,C 180,E1 -12491.24,E2 -12491.24} C_VEL
LIN {X 0,Y 381.969,Z 595.585,A -85,B 0,C 180,E1 -12491.703,E2 -12491.703} C_VEL
LIN {X 0,Y 381.352,Z 607.2,A -85,B 0,C 180,E1 -12492.297,E2 -12492.297} C_VEL
LIN {X 0,Y 380.524,Z 618.754,A -85,B 0,C 180,E1 -12493.089,E2 -12493.089} C_VEL
LIN {X 0,Y 379.606,Z 630.121,A -85,B 0,C 180,E1 -12494.095,E2 -12494.095} C_VEL
LIN {X 0,Y 378.757,Z 641.2,A -85,B 0,C 180,E1 -12495.356,E2 -12495.356} C_VEL
LIN {X 0,Y 377.597,Z 651.547,A -85,B 0,C 180,E1 -12496.82,E2 -12496.82} C_VEL
LIN {X 0,Y 376.836,Z 659.184,A -85,B 0,C 180,E1 -12498.162,E2 -12498.162} C_VEL
LIN {X 0,Y 376.112,Z 666.625,A -85,B 0,C 180,E1 -12499.775,E2 -12499.775} C_VEL
LIN {X 0,Y 375.44,Z 672.599,A -85,B 0,C 180,E1 -12501.387,E2 -12501.387} C_VEL
LIN {X 0,Y 375.079,Z 677.973,A -85,B 0,C 180,E1 -12503.259,E2 -12503.259} C_VEL
LIN {X 0,Y 374.849,Z 680.933,A -85,B 0,C 180,E1 -12504.621,E2 -12504.621} C_VEL
LIN {X 0,Y 374.67,Z 682.795,A -85,B 0,C 180,E1 -12505.697,E2 -12505.697} C_VEL
LIN {X 0,Y 374.567,Z 684.217,A -85,B 0,C 180,E1 -12506.773,E2 -12506.773} C_VEL
LIN {X 0,Y 374.545,Z 685.111,A -85,B 0,C 180,E1 -12507.741,E2 -12507.741} C_VEL
LIN {X 0,Y 373.895,Z 685.79,A -85,B 0,C 180,E1 -12508.633,E2 -12508.633} C_VEL
LIN {X 0,Y 372.31,Z 686.167,A -85,B 0,C 180,E1 -12509.511,E2 -12509.511} C_VEL
LIN {X 0,Y 368.576,Z 686.008,A -85,B 0,C 180,E1 -12511.272,E2 -12511.272} C_VEL
LIN {X 0,Y 367.529,Z 685.477,A -85,B 0,C 180,E1 -12512.181,E2 -12512.181} C_VEL
LIN {X 0,Y 367.446,Z 685.211,A -85,B 0,C 180,E1 -12512.488,E2 -12512.488} C_VEL
LIN {X 0,Y 367.604,Z 683.138,A -85,B 0,C 180,E1 -12514.386,E2 -12514.386} C_VEL
LIN {X 0,Y 367.871,Z 679.825,A -85,B 0,C 180,E1 -12516.235,E2 -12516.235} C_VEL
LIN {X 0,Y 368.27,Z 674.793,A -85,B 0,C 180,E1 -12518.229,E2 -12518.229} C_VEL
LIN {X 0,Y 368.833,Z 669.336,A -85,B 0,C 180,E1 -12519.875,E2 -12519.875} C_VEL
LIN {X 0,Y 369.575,Z 662.495,A -85,B 0,C 180,E1 -12521.518,E2 -12521.518} C_VEL
LIN {X 0,Y 370.468,Z 653.936,A -85,B 0,C 180,E1 -12523.159,E2 -12523.159} C_VEL
LIN {X 0,Y 371.481,Z 645.164,A -85,B 0,C 180,E1 -12524.518,E2 -12524.518} C_VEL
LIN {X 0,Y 372.335,Z 635.819,A -85,B 0,C 180,E1 -12525.708,E2 -12525.708} C_VEL
LIN {X 0,Y 373.175,Z 626.353,A -85,B 0,C 180,E1 -12526.691,E2 -12526.691} C_VEL
LIN {X 0,Y 374.072,Z 614.891,A -85,B 0,C 180,E1 -12527.635,E2 -12527.635} C_VEL
LIN {X 0,Y 374.966,Z 601.935,A -85,B 0,C 180,E1 -12528.439,E2 -12528.439} C_VEL
LIN {X 0,Y 375.461,Z 589.626,A -85,B 0,C 180,E1 -12528.98,E2 -12528.98} C_VEL
LIN {X 0,Y 375.956,Z 575.706,A -85,B 0,C 180,E1 -12529.343,E2 -12529.343} C_VEL
LIN {X 0,Y 377.116,Z 497.411,A -85,B 0,C 180,E1 -12530.845,E2 -12530.845} C_VEL
LIN {X 0,Y 372.722,Z 472.379,A -85,B 0,C 180,E1 -12531.625,E2 -12531.625} C_VEL
LIN {X 0,Y 373.389,Z 457.789,A -85,B 0,C 180,E1 -12534.166,E2 -12534.166} C_VEL
LIN {X 0,Y 373.787,Z 449.79,A -85,B 0,C 180,E1 -12535.623,E2 -12535.623} C_VEL
LIN {X 0,Y 371.225,Z 437.086,A -85,B 0,C 180,E1 -12538.249,E2 -12538.249} C_VEL
LIN {X 0,Y 368.923,Z 427.533,A -85,B 0,C 180,E1 -12540.32,E2 -12540.32} C_VEL
LIN {X 0,Y 368.899,Z 427.538,A -85,B 0,C 180,E1 -12543.538,E2 -12543.538} C_VEL
LIN {X 0,Y 368.903,Z 427.534,A -85,B 0,C 180,E1 -12546.856,E2 -12546.856} C_VEL
LIN {X 0,Y 368.913,Z 427.525,A -85,B 0,C 180,E1 -12550.37,E2 -12550.37} C_VEL
LIN {X 0,Y 368.885,Z 427.528,A -85,B 0,C 180,E1 -12553.616,E2 -12553.616} C_VEL
LIN {X 0,Y 368.889,Z 427.537,A -85,B 0,C 180,E1 -12556.696,E2 -12556.696} C_VEL
LIN {X 0,Y 368.914,Z 427.53,A -85,B 0,C 180,E1 -12559.643,E2 -12559.643} C_VEL
LIN {X 0,Y 368.903,Z 427.518,A -85,B 0,C 180,E1 -12563.144,E2 -12563.144} C_VEL
LIN {X 0,Y 368.899,Z 427.535,A -85,B 0,C 180,E1 -12566.462,E2 -12566.462} C_VEL
LIN {X 0,Y 368.924,Z 427.533,A -85,B 0,C 180,E1 -12570.31,E2 -12570.31} C_VEL
LIN {X 0,Y 368.968,Z 427.673,A -85,B 0,C 180,E1 -12570.886,E2 -12570.886} C_VEL
LIN {X 0,Y 372.516,Z 444.749,A -85,B 0,C 180,E1 -12574.283,E2 -12574.283} C_VEL
LIN {X 0,Y 373.003,Z 448.984,A -85,B 0,C 180,E1 -12575.094,E2 -12575.094} C_VEL
LIN {X 0,Y 372.146,Z 463.877,A -85,B 0,C 180,E1 -12577.808,E2 -12577.808} C_VEL
LIN {X 0,Y 371.701,Z 472.916,A -85,B 0,C 180,E1 -12579.451,E2 -12579.451} C_VEL
LIN {X 0,Y 375.001,Z 496.946,A -85,B 0,C 180,E1 -12580.216,E2 -12580.216} C_VEL
LIN {X 0,Y 372.987,Z 584.458,A -85,B 0,C 180,E1 -12582.383,E2 -12582.383} C_VEL
LIN {X 0,Y 372.429,Z 598.991,A -85,B 0,C 180,E1 -12582.992,E2 -12582.992} C_VEL
LIN {X 0,Y 371.708,Z 612.33,A -85,B 0,C 180,E1 -12583.806,E2 -12583.806} C_VEL
LIN {X 0,Y 371.097,Z 623.873,A -85,B 0,C 180,E1 -12584.728,E2 -12584.728} C_VEL
LIN {X 0,Y 370.45,Z 635.058,A -85,B 0,C 180,E1 -12585.862,E2 -12585.862} C_VEL
LIN {X 0,Y 369.774,Z 644.991,A -85,B 0,C 180,E1 -12587.096,E2 -12587.096} C_VEL
LIN {X 0,Y 369.101,Z 653.995,A -85,B 0,C 180,E1 -12588.467,E2 -12588.467} C_VEL
LIN {X 0,Y 368.498,Z 662.787,A -85,B 0,C 180,E1 -12590.116,E2 -12590.116} C_VEL
LIN {X 0,Y 368.022,Z 669.811,A -85,B 0,C 180,E1 -12591.765,E2 -12591.765} C_VEL
LIN {X 0,Y 367.719,Z 676.07,A -85,B 0,C 180,E1 -12593.642,E2 -12593.642} C_VEL
LIN {X 0,Y 367.625,Z 679.719,A -85,B 0,C 180,E1 -12595.065,E2 -12595.065} C_VEL
LIN {X 0,Y 367.446,Z 682.914,A -85,B 0,C 180,E1 -12596.711,E2 -12596.711} C_VEL
LIN {X 0,Y 367.418,Z 684.463,A -85,B 0,C 180,E1 -12597.807,E2 -12597.807} C_VEL
LIN {X 0,Y 367.412,Z 685.535,A -85,B 0,C 180,E1 -12598.904,E2 -12598.904} C_VEL
LIN {X 0,Y 367.44,Z 686.201,A -85,B 0,C 180,E1 -12600,E2 -12600} C_VEL
LIN {X 0,Y 367.467,Z 686.41,A -85,B 0,C 180,E1 -12601.096,E2 -12601.096} C_VEL
LIN {X 0,Y 367.511,Z 686.167,A -85,B 0,C 180,E1 -12602.192,E2 -12602.192} C_VEL
LIN {X 0,Y 367.53,Z 685.517,A -85,B 0,C 180,E1 -12603.289,E2 -12603.289} C_VEL
LIN {X 0,Y 367.614,Z 684.405,A -85,B 0,C 180,E1 -12604.386,E2 -12604.386} C_VEL
LIN {X 0,Y 367.878,Z 682.836,A -85,B 0,C 180,E1 -12605.481,E2 -12605.481} C_VEL
LIN {X 0,Y 368.067,Z 680.323,A -85,B 0,C 180,E1 -12606.826,E2 -12606.826} C_VEL
LIN {X 0,Y 368.629,Z 675.346,A -85,B 0,C 180,E1 -12608.773,E2 -12608.773} C_VEL
LIN {X 0,Y 369.289,Z 669.8,A -85,B 0,C 180,E1 -12610.416,E2 -12610.416} C_VEL
LIN {X 0,Y 370.077,Z 662.786,A -85,B 0,C 180,E1 -12612.058,E2 -12612.058} C_VEL
LIN {X 0,Y 371.181,Z 654.076,A -85,B 0,C 180,E1 -12613.69,E2 -12613.69} C_VEL
LIN {X 0,Y 372.196,Z 645.164,A -85,B 0,C 180,E1 -12615.048,E2 -12615.048} C_VEL
LIN {X 0,Y 373.433,Z 634.245,A -85,B 0,C 180,E1 -12616.398,E2 -12616.398} C_VEL
LIN {X 0,Y 374.55,Z 623.328,A -85,B 0,C 180,E1 -12617.471,E2 -12617.471} C_VEL
LIN {X 0,Y 375.677,Z 610.394,A -85,B 0,C 180,E1 -12618.473,E2 -12618.473} C_VEL
LIN {X 0,Y 376.694,Z 596.532,A -85,B 0,C 180,E1 -12619.269,E2 -12619.269} C_VEL
LIN {X 0,Y 377.441,Z 583.378,A -85,B 0,C 180,E1 -12619.795,E2 -12619.795} C_VEL
LIN {X 0,Y 381.157,Z 502.896,A -85,B 0,C 180,E1 -12622.067,E2 -12622.067} C_VEL
LIN {X 0,Y 381.169,Z 497.897,A -85,B 0,C 180,E1 -12622.239,E2 -12622.239} C_VEL
LIN {X 0,Y 378.444,Z 483.527,A -85,B 0,C 180,E1 -12623.024,E2 -12623.024} C_VEL
LIN {X 0,Y 376.422,Z 475.193,A -85,B 0,C 180,E1 -12623.574,E2 -12623.574} C_VEL
LIN {X 0,Y 377.869,Z 459.686,A -85,B 0,C 180,E1 -12626.511,E2 -12626.511} C_VEL
LIN {X 0,Y 377.219,Z 454.09,A -85,B 0,C 180,E1 -12627.761,E2 -12627.761} C_VEL
LIN {X 0,Y 375.24,Z 445.54,A -85,B 0,C 180,E1 -12629.856,E2 -12629.856} C_VEL
LIN {X 0,Y 372.184,Z 436.175,A -85,B 0,C 180,E1 -12632.473,E2 -12632.473} C_VEL
LIN {X 0,Y 369.981,Z 430.476,A -85,B 0,C 180,E1 -12634.253,E2 -12634.253} C_VEL
LIN {X 0,Y 368.938,Z 427.529,A -85,B 0,C 180,E1 -12635.265,E2 -12635.265} C_VEL
LIN {X 0,Y 368.905,Z 427.534,A -85,B 0,C 180,E1 -12638.953,E2 -12638.953} C_VEL
LIN {X 0,Y 368.883,Z 427.535,A -85,B 0,C 180,E1 -12642.009,E2 -12642.009} C_VEL
LIN {X 0,Y 368.882,Z 427.533,A -85,B 0,C 180,E1 -12645.176,E2 -12645.176} C_VEL
LIN {X 0,Y 368.885,Z 427.537,A -85,B 0,C 180,E1 -12648.178,E2 -12648.178} C_VEL
LIN {X 0,Y 368.91,Z 427.53,A -85,B 0,C 180,E1 -12651.36,E2 -12651.36} C_VEL
LIN {X 0,Y 368.938,Z 427.528,A -85,B 0,C 180,E1 -12655.146,E2 -12655.146} C_VEL
LIN {X 0,Y 368.951,Z 427.674,A -85,B 0,C 180,E1 -12658.052,E2 -12658.052} C_VEL
LIN {X 0,Y 372.511,Z 444.452,A -85,B 0,C 180,E1 -12661.551,E2 -12661.551} C_VEL
LIN {X 0,Y 373.373,Z 449.781,A -85,B 0,C 180,E1 -12662.619,E2 -12662.619} C_VEL
LIN {X 0,Y 372.681,Z 458.474,A -85,B 0,C 180,E1 -12664.22,E2 -12664.22} C_VEL
LIN {X 0,Y 374.125,Z 474.202,A -85,B 0,C 180,E1 -12665.737,E2 -12665.737} C_VEL
LIN {X 0,Y 375.153,Z 485.101,A -85,B 0,C 180,E1 -12666.629,E2 -12666.629} C_VEL
LIN {X 0,Y 377.606,Z 501.568,A -85,B 0,C 180,E1 -12667.515,E2 -12667.515} C_VEL
LIN {X 0,Y 378.647,Z 513.543,A -85,B 0,C 180,E1 -12668.044,E2 -12668.044} C_VEL
LIN {X 0,Y 379.415,Z 525.379,A -85,B 0,C 180,E1 -12668.535,E2 -12668.535} C_VEL
LIN {X 0,Y 375.521,Z 607.568,A -85,B 0,C 180,E1 -12670.917,E2 -12670.917} C_VEL
LIN {X 0,Y 374.673,Z 621.506,A -85,B 0,C 180,E1 -12671.546,E2 -12671.546} C_VEL
LIN {X 0,Y 373.678,Z 634.137,A -85,B 0,C 180,E1 -12672.346,E2 -12672.346} C_VEL
LIN {X 0,Y 372.612,Z 645.566,A -85,B 0,C 180,E1 -12673.283,E2 -12673.283} C_VEL
LIN {X 0,Y 371.543,Z 657.124,A -85,B 0,C 180,E1 -12674.503,E2 -12674.503} C_VEL
LIN {X 0,Y 370.553,Z 666.558,A -85,B 0,C 180,E1 -12675.726,E2 -12675.726} C_VEL
LIN {X 0,Y 369.704,Z 675.212,A -85,B 0,C 180,E1 -12677.093,E2 -12677.093} C_VEL
LIN {X 0,Y 368.855,Z 683.655,A -85,B 0,C 180,E1 -12678.738,E2 -12678.738} C_VEL
LIN {X 0,Y 368.263,Z 690.416,A -85,B 0,C 180,E1 -12680.387,E2 -12680.387} C_VEL
LIN {X 0,Y 367.752,Z 696.485,A -85,B 0,C 180,E1 -12682.312,E2 -12682.312} C_VEL
LIN {X 0,Y 367.577,Z 700.153,A -85,B 0,C 180,E1 -12683.844,E2 -12683.844} C_VEL
LIN {X 0,Y 367.533,Z 703.2,A -85,B 0,C 180,E1 -12685.613,E2 -12685.613} C_VEL
LIN {X 0,Y 367.446,Z 704.485,A -85,B 0,C 180,E1 -12686.711,E2 -12686.711} C_VEL
LIN {X 0,Y 367.428,Z 705.279,A -85,B 0,C 180,E1 -12687.808,E2 -12687.808} C_VEL
LIN {X 0,Y 367.532,Z 705.826,A -85,B 0,C 180,E1 -12690,E2 -12690} C_VEL
LIN {X 0,Y 367.477,Z 705.601,A -85,B 0,C 180,E1 -12691.096,E2 -12691.096} C_VEL
LIN {X 0,Y 367.451,Z 703.972,A -85,B 0,C 180,E1 -12693.289,E2 -12693.289} C_VEL
LIN {X 0,Y 367.512,Z 702.539,A -85,B 0,C 180,E1 -12694.387,E2 -12694.387} C_VEL
LIN {X 0,Y 367.568,Z 699.312,A -85,B 0,C 180,E1 -12696.144,E2 -12696.144} C_VEL
LIN {X 0,Y 367.76,Z 695.504,A -85,B 0,C 180,E1 -12697.688,E2 -12697.688} C_VEL
LIN {X 0,Y 368.199,Z 689.259,A -85,B 0,C 180,E1 -12699.614,E2 -12699.614} C_VEL
LIN {X 0,Y 368.767,Z 682.445,A -85,B 0,C 180,E1 -12701.265,E2 -12701.265} C_VEL
LIN {X 0,Y 369.501,Z 675.473,A -85,B 0,C 180,E1 -12702.635,E2 -12702.635} C_VEL
LIN {X 0,Y 370.266,Z 667.044,A -85,B 0,C 180,E1 -12704.005,E2 -12704.005} C_VEL
LIN {X 0,Y 371.248,Z 656.61,A -85,B 0,C 180,E1 -12705.369,E2 -12705.369} C_VEL
LIN {X 0,Y 372.208,Z 646.27,A -85,B 0,C 180,E1 -12706.453,E2 -12706.453} C_VEL
LIN {X 0,Y 373.174,Z 634.875,A -85,B 0,C 180,E1 -12707.396,E2 -12707.396} C_VEL
LIN {X 0,Y 374.015,Z 623.051,A -85,B 0,C 180,E1 -12708.133,E2 -12708.133} C_VEL
LIN {X 0,Y 374.461,Z 616.776,A -85,B 0,C 180,E1 -12708.464,E2 -12708.464} C_VEL
LIN {X 0,Y 375.808,Z 603.087,A -85,B 0,C 180,E1 -12709.245,E2 -12709.245} C_VEL
LIN {X 0,Y 376.854,Z 588.661,A -85,B 0,C 180,E1 -12709.827,E2 -12709.827} C_VEL
LIN {X 0,Y 379.493,Z 523.614,A -85,B 0,C 180,E1 -12711.657,E2 -12711.657} C_VEL
LIN {X 0,Y 378.079,Z 505.373,A -85,B 0,C 180,E1 -12712.402,E2 -12712.402} C_VEL
LIN {X 0,Y 375.387,Z 487.267,A -85,B 0,C 180,E1 -12713.31,E2 -12713.31} C_VEL
LIN {X 0,Y 373.034,Z 475.284,A -85,B 0,C 180,E1 -12714.043,E2 -12714.043} C_VEL
LIN {X 0,Y 375.484,Z 457.118,A -85,B 0,C 180,E1 -12717.9,E2 -12717.9} C_VEL
LIN {X 0,Y 375.547,Z 453.885,A -85,B 0,C 180,E1 -12718.656,E2 -12718.656} C_VEL
LIN {X 0,Y 374.309,Z 447.176,A -85,B 0,C 180,E1 -12720.461,E2 -12720.461} C_VEL
LIN {X 0,Y 372.129,Z 438.165,A -85,B 0,C 180,E1 -12723.209,E2 -12723.209} C_VEL
LIN {X 0,Y 369.799,Z 430.215,A -85,B 0,C 180,E1 -12726.097,E2 -12726.097} C_VEL
LIN {X 0,Y 368.898,Z 427.535,A -85,B 0,C 180,E1 -12727.264,E2 -12727.264} C_VEL
LIN {X 0,Y 368.911,Z 427.534,A -85,B 0,C 180,E1 -12730.37,E2 -12730.37} C_VEL
LIN {X 0,Y 368.884,Z 427.535,A -85,B 0,C 180,E1 -12733.616,E2 -12733.616} C_VEL
LIN {X 0,Y 368.887,Z 427.534,A -85,B 0,C 180,E1 -12736.696,E2 -12736.696} C_VEL
LIN {X 0,Y 368.913,Z 427.531,A -85,B 0,C 180,E1 -12739.643,E2 -12739.643} C_VEL
LIN {X 0,Y 368.903,Z 427.532,A -85,B 0,C 180,E1 -12743.144,E2 -12743.144} C_VEL
LIN {X 0,Y 368.898,Z 427.533,A -85,B 0,C 180,E1 -12746.462,E2 -12746.462} C_VEL
LIN {X 0,Y 368.931,Z 427.53,A -85,B 0,C 180,E1 -12749.047,E2 -12749.047} C_VEL
LIN {X 0,Y 368.965,Z 427.528,A -85,B 0,C 180,E1 -12752.797,E2 -12752.797} C_VEL
LIN {X 0,Y 368.967,Z 427.617,A -85,B 0,C 180,E1 -12755,E2 -12755} C_VEL
LIN {X 0,Y 369.306,Z 429.019,A -85,B 0,C 180,E1 -12755.654,E2 -12755.654} C_VEL
LIN {X 0,Y 372.122,Z 433.833,A -85,B 0,C 180,E1 -12756.218,E2 -12756.218} C_VEL
LIN {X 0,Y 376.429,Z 441.304,A -85,B 0,C 180,E1 -12757.029,E2 -12757.029} C_VEL
LIN {X 0,Y 381.457,Z 451.407,A -85,B 0,C 180,E1 -12757.956,E2 -12757.956} C_VEL
LIN {X 0,Y 381.914,Z 452.935,A -85,B 0,C 180,E1 -12758.058,E2 -12758.058} C_VEL
LIN {X 0,Y 378.615,Z 518.623,A -85,B 0,C 180,E1 -12759.951,E2 -12759.951} C_VEL
LIN {X 0,Y 378.029,Z 535,A -85,B 0,C 180,E1 -12760.485,E2 -12760.485} C_VEL
LIN {X 0,Y 377.442,Z 547.662,A -85,B 0,C 180,E1 -12761.124,E2 -12761.124} C_VEL
LIN {X 0,Y 376.691,Z 559.575,A -85,B 0,C 180,E1 -12761.931,E2 -12761.931} C_VEL
LIN {X 0,Y 375.658,Z 571.414,A -85,B 0,C 180,E1 -12762.955,E2 -12762.955} C_VEL
LIN {X 0,Y 374.48,Z 582.87,A -85,B 0,C 180,E1 -12764.209,E2 -12764.209} C_VEL
LIN {X 0,Y 373.394,Z 592.652,A -85,B 0,C 180,E1 -12765.559,E2 -12765.559} C_VEL
LIN {X 0,Y 372.247,Z 602.072,A -85,B 0,C 180,E1 -12767.183,E2 -12767.183} C_VEL
LIN {X 0,Y 371.194,Z 609.591,A -85,B 0,C 180,E1 -12768.81,E2 -12768.81} C_VEL
LIN {X 0,Y 370.542,Z 614.705,A -85,B 0,C 180,E1 -12770.171,E2 -12770.171} C_VEL
LIN {X 0,Y 369.797,Z 619.611,A -85,B 0,C 180,E1 -12771.805,E2 -12771.805} C_VEL
LIN {X 0,Y 369.173,Z 623.345,A -85,B 0,C 180,E1 -12773.441,E2 -12773.441} C_VEL
LIN {X 0,Y 368.935,Z 625.206,A -85,B 0,C 180,E1 -12774.534,E2 -12774.534} C_VEL
LIN {X 0,Y 368.633,Z 626.654,A -85,B 0,C 180,E1 -12775.626,E2 -12775.626} C_VEL
LIN {X 0,Y 368.301,Z 627.656,A -85,B 0,C 180,E1 -12776.718,E2 -12776.718} C_VEL
LIN {X 0,Y 368.061,Z 628.203,A -85,B 0,C 180,E1 -12777.811,E2 -12777.811} C_VEL
LIN {X 0,Y 367.936,Z 628.336,A -85,B 0,C 180,E1 -12778.906,E2 -12778.906} C_VEL
LIN {X 0,Y 367.889,Z 628.047,A -85,B 0,C 180,E1 -12780,E2 -12780} C_VEL
LIN {X 0,Y 367.916,Z 627.288,A -85,B 0,C 180,E1 -12781.095,E2 -12781.095} C_VEL
LIN {X 0,Y 368.022,Z 626.109,A -85,B 0,C 180,E1 -12782.189,E2 -12782.189} C_VEL
LIN {X 0,Y 368.208,Z 623.52,A -85,B 0,C 180,E1 -12783.831,E2 -12783.831} C_VEL
LIN {X 0,Y 368.352,Z 619.891,A -85,B 0,C 180,E1 -12785.474,E2 -12785.474} C_VEL
LIN {X 0,Y 368.578,Z 614.902,A -85,B 0,C 180,E1 -12787.183,E2 -12787.183} C_VEL
LIN {X 0,Y 368.881,Z 609.053,A -85,B 0,C 180,E1 -12788.767,E2 -12788.767} C_VEL
LIN {X 0,Y 369.44,Z 601.439,A -85,B 0,C 180,E1 -12790.412,E2 -12790.412} C_VEL
LIN {X 0,Y 370.036,Z 591.987,A -85,B 0,C 180,E1 -12792.059,E2 -12792.059} C_VEL
LIN {X 0,Y 370.715,Z 582.213,A -85,B 0,C 180,E1 -12793.429,E2 -12793.429} C_VEL
LIN {X 0,Y 371.328,Z 571.495,A -85,B 0,C 180,E1 -12794.652,E2 -12794.652} C_VEL
LIN {X 0,Y 371.993,Z 560.049,A -85,B 0,C 180,E1 -12795.704,E2 -12795.704} C_VEL
LIN {X 0,Y 372.453,Z 547.809,A -85,B 0,C 180,E1 -12796.583,E2 -12796.583} C_VEL
LIN {X 0,Y 372.983,Z 534.461,A -85,B 0,C 180,E1 -12797.299,E2 -12797.299} C_VEL
LIN {X 0,Y 373.317,Z 521.301,A -85,B 0,C 180,E1 -12797.778,E2 -12797.778} C_VEL
LIN {X 0,Y 374.988,Z 445.716,A -85,B 0,C 180,E1 -12799.648,E2 -12799.648} C_VEL
LIN {X 0,Y 368.981,Z 427.527,A -85,B 0,C 180,E1 -12800.383,E2 -12800.383} C_VEL
LIN {X 0,Y 368.935,Z 427.526,A -85,B 0,C 180,E1 -12803.883,E2 -12803.883} C_VEL
LIN {X 0,Y 368.965,Z 427.521,A -85,B 0,C 180,E1 -12807.203,E2 -12807.203} C_VEL
LIN {X 0,Y 368.931,Z 427.529,A -85,B 0,C 180,E1 -12810.954,E2 -12810.954} C_VEL
LIN {X 0,Y 368.931,Z 427.515,A -85,B 0,C 180,E1 -12815.001,E2 -12815.001} C_VEL
LIN {X 0,Y 368.91,Z 427.532,A -85,B 0,C 180,E1 -12818.64,E2 -12818.64} C_VEL
LIN {X 0,Y 368.884,Z 427.532,A -85,B 0,C 180,E1 -12822.009,E2 -12822.009} C_VEL
LIN {X 0,Y 368.882,Z 427.525,A -85,B 0,C 180,E1 -12825.176,E2 -12825.176} C_VEL
LIN {X 0,Y 368.885,Z 427.535,A -85,B 0,C 180,E1 -12828.178,E2 -12828.178} C_VEL
LIN {X 0,Y 368.91,Z 427.533,A -85,B 0,C 180,E1 -12831.36,E2 -12831.36} C_VEL
LIN {X 0,Y 368.939,Z 427.528,A -85,B 0,C 180,E1 -12835.147,E2 -12835.147} C_VEL
LIN {X 0,Y 368.931,Z 427.534,A -85,B 0,C 180,E1 -12839.047,E2 -12839.047} C_VEL
LIN {X 0,Y 368.947,Z 427.544,A -85,B 0,C 180,E1 -12839.84,E2 -12839.84} C_VEL
LIN {X 0,Y 371.97,Z 440.703,A -85,B 0,C 180,E1 -12842.626,E2 -12842.626} C_VEL
LIN {X 0,Y 373.799,Z 449.757,A -85,B 0,C 180,E1 -12844.486,E2 -12844.486} C_VEL
LIN {X 0,Y 373.052,Z 464.659,A -85,B 0,C 180,E1 -12847.167,E2 -12847.167} C_VEL
LIN {X 0,Y 372.703,Z 472.386,A -85,B 0,C 180,E1 -12848.48,E2 -12848.48} C_VEL
LIN {X 0,Y 377.08,Z 497.689,A -85,B 0,C 180,E1 -12849.26,E2 -12849.26} C_VEL
LIN {X 0,Y 375.767,Z 579.252,A -85,B 0,C 180,E1 -12850.824,E2 -12850.824} C_VEL
LIN {X 0,Y 375.379,Z 592.407,A -85,B 0,C 180,E1 -12851.229,E2 -12851.229} C_VEL
LIN {X 0,Y 374.696,Z 605.061,A -85,B 0,C 180,E1 -12851.831,E2 -12851.831} C_VEL
LIN {X 0,Y 373.867,Z 617.241,A -85,B 0,C 180,E1 -12852.637,E2 -12852.637} C_VEL
LIN {X 0,Y 372.864,Z 629.296,A -85,B 0,C 180,E1 -12853.697,E2 -12853.697} C_VEL
LIN {X 0,Y 371.999,Z 640.348,A -85,B 0,C 180,E1 -12854.943,E2 -12854.943} C_VEL
LIN {X 0,Y 370.921,Z 649.999,A -85,B 0,C 180,E1 -12856.3,E2 -12856.3} C_VEL
LIN {X 0,Y 370.003,Z 657.928,A -85,B 0,C 180,E1 -12857.661,E2 -12857.661} C_VEL
LIN {X 0,Y 369.205,Z 665.7,A -85,B 0,C 180,E1 -12859.304,E2 -12859.304} C_VEL
LIN {X 0,Y 368.635,Z 670.951,A -85,B 0,C 180,E1 -12860.674,E2 -12860.674} C_VEL
LIN {X 0,Y 368.112,Z 676.083,A -85,B 0,C 180,E1 -12862.32,E2 -12862.32} C_VEL
LIN {X 0,Y 367.879,Z 679.583,A -85,B 0,C 180,E1 -12863.755,E2 -12863.755} C_VEL
LIN {X 0,Y 367.605,Z 682.984,A -85,B 0,C 180,E1 -12865.614,E2 -12865.614} C_VEL
LIN {X 0,Y 367.482,Z 684.406,A -85,B 0,C 180,E1 -12866.711,E2 -12866.711} C_VEL
LIN {X 0,Y 367.447,Z 686.014,A -85,B 0,C 180,E1 -12868.904,E2 -12868.904} C_VEL
LIN {X 0,Y 367.441,Z 686.249,A -85,B 0,C 180,E1 -12870,E2 -12870} C_VEL
LIN {X 0,Y 367.447,Z 686.057,A -85,B 0,C 180,E1 -12871.096,E2 -12871.096} C_VEL
LIN {X 0,Y 367.446,Z 685.211,A -85,B 0,C 180,E1 -12872.488,E2 -12872.488} C_VEL
LIN {X 0,Y 366.809,Z 684.423,A -85,B 0,C 180,E1 -12873.395,E2 -12873.395} C_VEL
LIN {X 0,Y 364.09,Z 682.552,A -85,B 0,C 180,E1 -12874.863,E2 -12874.863} C_VEL
LIN {X 0,Y 361.85,Z 680.615,A -85,B 0,C 180,E1 -12876.033,E2 -12876.033} C_VEL
LIN {X 0,Y 360.975,Z 678.792,A -85,B 0,C 180,E1 -12876.92,E2 -12876.92} C_VEL
LIN {X 0,Y 360.95,Z 678.076,A -85,B 0,C 180,E1 -12877.216,E2 -12877.216} C_VEL
LIN {X 0,Y 361.387,Z 673.293,A -85,B 0,C 180,E1 -12878.95,E2 -12878.95} C_VEL
LIN {X 0,Y 362.048,Z 667.388,A -85,B 0,C 180,E1 -12880.627,E2 -12880.627} C_VEL
LIN {X 0,Y 362.886,Z 660.041,A -85,B 0,C 180,E1 -12882.3,E2 -12882.3} C_VEL
LIN {X 0,Y 363.798,Z 652.528,A -85,B 0,C 180,E1 -12883.689,E2 -12883.689} C_VEL
LIN {X 0,Y 364.948,Z 642.316,A -85,B 0,C 180,E1 -12885.212,E2 -12885.212} C_VEL
LIN {X 0,Y 365.842,Z 631.962,A -85,B 0,C 180,E1 -12886.46,E2 -12886.46} C_VEL
LIN {X 0,Y 366.799,Z 621.971,A -85,B 0,C 180,E1 -12887.42,E2 -12887.42} C_VEL
LIN {X 0,Y 367.684,Z 610.13,A -85,B 0,C 180,E1 -12888.312,E2 -12888.312} C_VEL
LIN {X 0,Y 368.474,Z 597.24,A -85,B 0,C 180,E1 -12889.028,E2 -12889.028} C_VEL
LIN {X 0,Y 368.926,Z 585.655,A -85,B 0,C 180,E1 -12889.474,E2 -12889.474} C_VEL
LIN {X 0,Y 369.497,Z 561.519,A -85,B 0,C 180,E1 -12889.985,E2 -12889.985} C_VEL
LIN {X 0,Y 370.362,Z 497.254,A -85,B 0,C 180,E1 -12891.247,E2 -12891.247} C_VEL
LIN {X 0,Y 365.912,Z 472.572,A -85,B 0,C 180,E1 -12892.034,E2 -12892.034} C_VEL
LIN {X 0,Y 366.823,Z 456.211,A -85,B 0,C 180,E1 -12894.929,E2 -12894.929} C_VEL
LIN {X 0,Y 366.958,Z 451.365,A -85,B 0,C 180,E1 -12895.822,E2 -12895.822} C_VEL
LIN {X 0,Y 364.342,Z 438.504,A -85,B 0,C 180,E1 -12898.517,E2 -12898.517} C_VEL
LIN {X 0,Y 361.878,Z 428.41,A -85,B 0,C 180,E1 -12900.709,E2 -12900.709} C_VEL
LIN {X 0,Y 361.857,Z 428.415,A -85,B 0,C 180,E1 -12904.28,E2 -12904.28} C_VEL
LIN {X 0,Y 361.865,Z 428.408,A -85,B 0,C 180,E1 -12907.223,E2 -12907.223} C_VEL
LIN {X 0,Y 361.838,Z 428.407,A -85,B 0,C 180,E1 -12910.755,E2 -12910.755} C_VEL
LIN {X 0,Y 361.823,Z 428.409,A -85,B 0,C 180,E1 -12914.368,E2 -12914.368} C_VEL
LIN {X 0,Y 361.839,Z 428.405,A -85,B 0,C 180,E1 -12917.568,E2 -12917.568} C_VEL
LIN {X 0,Y 361.872,Z 428.411,A -85,B 0,C 180,E1 -12920.973,E2 -12920.973} C_VEL
LIN {X 0,Y 361.876,Z 428.398,A -85,B 0,C 180,E1 -12924.655,E2 -12924.655} C_VEL
LIN {X 0,Y 361.84,Z 428.415,A -85,B 0,C 180,E1 -12928.371,E2 -12928.371} C_VEL
LIN {X 0,Y 361.905,Z 428.474,A -85,B 0,C 180,E1 -12930.625,E2 -12930.625} C_VEL
LIN {X 0,Y 365.409,Z 445.234,A -85,B 0,C 180,E1 -12933.998,E2 -12933.998} C_VEL
LIN {X 0,Y 366.045,Z 450.451,A -85,B 0,C 180,E1 -12935.014,E2 -12935.014} C_VEL
LIN {X 0,Y 365.033,Z 468.107,A -85,B 0,C 180,E1 -12938.262,E2 -12938.262} C_VEL
LIN {X 0,Y 364.789,Z 473.106,A -85,B 0,C 180,E1 -12939.178,E2 -12939.178} C_VEL
LIN {X 0,Y 368.1,Z 498.195,A -85,B 0,C 180,E1 -12939.981,E2 -12939.981} C_VEL
LIN {X 0,Y 366.007,Z 584.197,A -85,B 0,C 180,E1 -12942.18,E2 -12942.18} C_VEL
LIN {X 0,Y 365.456,Z 598.77,A -85,B 0,C 180,E1 -12942.802,E2 -12942.802} C_VEL
LIN {X 0,Y 364.71,Z 612.195,A -85,B 0,C 180,E1 -12943.631,E2 -12943.631} C_VEL
LIN {X 0,Y 364.089,Z 623.577,A -85,B 0,C 180,E1 -12944.549,E2 -12944.549} C_VEL
LIN {X 0,Y 363.417,Z 635.047,A -85,B 0,C 180,E1 -12945.725,E2 -12945.725} C_VEL
LIN {X 0,Y 362.645,Z 646.015,A -85,B 0,C 180,E1 -12947.122,E2 -12947.122} C_VEL
LIN {X 0,Y 361.831,Z 656.482,A -85,B 0,C 180,E1 -12948.8,E2 -12948.8} C_VEL
LIN {X 0,Y 361.298,Z 664.801,A -85,B 0,C 180,E1 -12950.483,E2 -12950.483} C_VEL
LIN {X 0,Y 360.852,Z 671.495,A -85,B 0,C 180,E1 -12952.164,E2 -12952.164} C_VEL
LIN {X 0,Y 360.634,Z 676.259,A -85,B 0,C 180,E1 -12953.662,E2 -12953.662} C_VEL
LIN {X 0,Y 360.496,Z 680.822,A -85,B 0,C 180,E1 -12955.527,E2 -12955.527} C_VEL
LIN {X 0,Y 360.367,Z 682.884,A -85,B 0,C 180,E1 -12956.646,E2 -12956.646} C_VEL
LIN {X 0,Y 360.321,Z 684.511,A -85,B 0,C 180,E1 -12957.764,E2 -12957.764} C_VEL
LIN {X 0,Y 360.313,Z 685.64,A -85,B 0,C 180,E1 -12958.882,E2 -12958.882} C_VEL
LIN {X 0,Y 360.342,Z 686.347,A -85,B 0,C 180,E1 -12960,E2 -12960} C_VEL
LIN {X 0,Y 360.371,Z 686.63,A -85,B 0,C 180,E1 -12961.117,E2 -12961.117} C_VEL
LIN {X 0,Y 360.416,Z 686.435,A -85,B 0,C 180,E1 -12962.235,E2 -12962.235} C_VEL
LIN {X 0,Y 360.444,Z 685.83,A -85,B 0,C 180,E1 -12963.353,E2 -12963.353} C_VEL
LIN {X 0,Y 360.556,Z 684.8,A -85,B 0,C 180,E1 -12964.472,E2 -12964.472} C_VEL
LIN {X 0,Y 360.831,Z 683.28,A -85,B 0,C 180,E1 -12965.589,E2 -12965.589} C_VEL
LIN {X 0,Y 361.106,Z 680.176,A -85,B 0,C 180,E1 -12967.267,E2 -12967.267} C_VEL
LIN {X 0,Y 361.627,Z 675.942,A -85,B 0,C 180,E1 -12968.944,E2 -12968.944} C_VEL
LIN {X 0,Y 362.344,Z 670.491,A -85,B 0,C 180,E1 -12970.618,E2 -12970.618} C_VEL
LIN {X 0,Y 363.195,Z 663.659,A -85,B 0,C 180,E1 -12972.29,E2 -12972.29} C_VEL
LIN {X 0,Y 364.387,Z 655.111,A -85,B 0,C 180,E1 -12973.951,E2 -12973.951} C_VEL
LIN {X 0,Y 365.457,Z 646.389,A -85,B 0,C 180,E1 -12975.333,E2 -12975.333} C_VEL
LIN {X 0,Y 366.749,Z 635.627,A -85,B 0,C 180,E1 -12976.705,E2 -12976.705} C_VEL
LIN {X 0,Y 367.941,Z 625.135,A -85,B 0,C 180,E1 -12977.795,E2 -12977.795} C_VEL
LIN {X 0,Y 369.049,Z 613.664,A -85,B 0,C 180,E1 -12978.745,E2 -12978.745} C_VEL
LIN {X 0,Y 370.096,Z 601.09,A -85,B 0,C 180,E1 -12979.554,E2 -12979.554} C_VEL
LIN {X 0,Y 371.034,Z 587.162,A -85,B 0,C 180,E1 -12980.188,E2 -12980.188} C_VEL
LIN {X 0,Y 375.381,Z 500.093,A -85,B 0,C 180,E1 -12982.762,E2 -12982.762} C_VEL
LIN {X 0,Y 372.823,Z 486.013,A -85,B 0,C 180,E1 -12983.569,E2 -12983.569} C_VEL
LIN {X 0,Y 370.306,Z 475.37,A -85,B 0,C 180,E1 -12984.313,E2 -12984.313} C_VEL
LIN {X 0,Y 371.634,Z 461.609,A -85,B 0,C 180,E1 -12986.992,E2 -12986.992} C_VEL
LIN {X 0,Y 370.496,Z 454.325,A -85,B 0,C 180,E1 -12988.729,E2 -12988.729} C_VEL
LIN {X 0,Y 368.988,Z 448.211,A -85,B 0,C 180,E1 -12990.325,E2 -12990.325} C_VEL
LIN {X 0,Y 366.64,Z 440.696,A -85,B 0,C 180,E1 -12992.496,E2 -12992.496} C_VEL
LIN {X 0,Y 364.242,Z 434.319,A -85,B 0,C 180,E1 -12994.591,E2 -12994.591} C_VEL
LIN {X 0,Y 363.066,Z 431.512,A -85,B 0,C 180,E1 -12995.609,E2 -12995.609} C_VEL
LIN {X 0,Y 361.873,Z 428.408,A -85,B 0,C 180,E1 -12996.843,E2 -12996.843} C_VEL
LIN {X 0,Y 361.857,Z 428.408,A -85,B 0,C 180,E1 -12999.861,E2 -12999.861} C_VEL
LIN {X 0,Y 361.838,Z 428.412,A -85,B 0,C 180,E1 -13002.829,E2 -13002.829} C_VEL
LIN {X 0,Y 361.82,Z 428.417,A -85,B 0,C 180,E1 -13005.946,E2 -13005.946} C_VEL
LIN {X 0,Y 361.837,Z 428.41,A -85,B 0,C 180,E1 -13009.245,E2 -13009.245} C_VEL
LIN {X 0,Y 361.865,Z 428.405,A -85,B 0,C 180,E1 -13012.777,E2 -13012.777} C_VEL
LIN {X 0,Y 361.856,Z 428.41,A -85,B 0,C 180,E1 -13015.72,E2 -13015.72} C_VEL
LIN {X 0,Y 361.903,Z 428.478,A -85,B 0,C 180,E1 -13017.803,E2 -13017.803} C_VEL
LIN {X 0,Y 365.59,Z 445.942,A -85,B 0,C 180,E1 -13021.511,E2 -13021.511} C_VEL
LIN {X 0,Y 366.301,Z 449.739,A -85,B 0,C 180,E1 -13022.286,E2 -13022.286} C_VEL
LIN {X 0,Y 367.263,Z 462.043,A -85,B 0,C 180,E1 -13023.735,E2 -13023.735} C_VEL
LIN {X 0,Y 368.521,Z 478.194,A -85,B 0,C 180,E1 -13025.343,E2 -13025.343} C_VEL
LIN {X 0,Y 369.143,Z 484.884,A -85,B 0,C 180,E1 -13025.904,E2 -13025.904} C_VEL
LIN {X 0,Y 371.548,Z 500.743,A -85,B 0,C 180,E1 -13026.813,E2 -13026.813} C_VEL
LIN {X 0,Y 372.643,Z 513.114,A -85,B 0,C 180,E1 -13027.408,E2 -13027.408} C_VEL
LIN {X 0,Y 373.386,Z 526.507,A -85,B 0,C 180,E1 -13027.971,E2 -13027.971} C_VEL
LIN {X 0,Y 369.898,Z 595.599,A -85,B 0,C 180,E1 -13030.037,E2 -13030.037} C_VEL
LIN {X 0,Y 369.092,Z 610.72,A -85,B 0,C 180,E1 -13030.535,E2 -13030.535} C_VEL
LIN {X 0,Y 368.097,Z 624,A -85,B 0,C 180,E1 -13031.204,E2 -13031.204} C_VEL
LIN {X 0,Y 367.038,Z 635.883,A -85,B 0,C 180,E1 -13032.015,E2 -13032.015} C_VEL
LIN {X 0,Y 365.912,Z 646.762,A -85,B 0,C 180,E1 -13032.968,E2 -13032.968} C_VEL
LIN {X 0,Y 364.862,Z 656.943,A -85,B 0,C 180,E1 -13034.069,E2 -13034.069} C_VEL
LIN {X 0,Y 363.729,Z 667.297,A -85,B 0,C 180,E1 -13035.452,E2 -13035.452} C_VEL
LIN {X 0,Y 362.667,Z 677.262,A -85,B 0,C 180,E1 -13037.123,E2 -13037.123} C_VEL
LIN {X 0,Y 361.779,Z 685.214,A -85,B 0,C 180,E1 -13038.798,E2 -13038.798} C_VEL
LIN {X 0,Y 361.177,Z 691.602,A -85,B 0,C 180,E1 -13040.48,E2 -13040.48} C_VEL
LIN {X 0,Y 360.695,Z 696.637,A -85,B 0,C 180,E1 -13042.161,E2 -13042.161} C_VEL
LIN {X 0,Y 360.494,Z 700.494,A -85,B 0,C 180,E1 -13043.864,E2 -13043.864} C_VEL
LIN {X 0,Y 360.436,Z 703.162,A -85,B 0,C 180,E1 -13045.527,E2 -13045.527} C_VEL
LIN {X 0,Y 360.364,Z 704.372,A -85,B 0,C 180,E1 -13046.646,E2 -13046.646} C_VEL
LIN {X 0,Y 360.33,Z 705.132,A -85,B 0,C 180,E1 -13047.764,E2 -13047.764} C_VEL
LIN {X 0,Y 360.434,Z 705.637,A -85,B 0,C 180,E1 -13050,E2 -13050} C_VEL
LIN {X 0,Y 360.376,Z 705.412,A -85,B 0,C 180,E1 -13051.117,E2 -13051.117} C_VEL
LIN {X 0,Y 360.367,Z 703.783,A -85,B 0,C 180,E1 -13053.354,E2 -13053.354} C_VEL
LIN {X 0,Y 360.417,Z 702.349,A -85,B 0,C 180,E1 -13054.474,E2 -13054.474} C_VEL
LIN {X 0,Y 360.462,Z 699.508,A -85,B 0,C 180,E1 -13056.088,E2 -13056.088} C_VEL
LIN {X 0,Y 360.7,Z 695.315,A -85,B 0,C 180,E1 -13057.839,E2 -13057.839} C_VEL
LIN {X 0,Y 361.173,Z 689.07,A -85,B 0,C 180,E1 -13059.803,E2 -13059.803} C_VEL
LIN {X 0,Y 361.784,Z 682.257,A -85,B 0,C 180,E1 -13061.485,E2 -13061.485} C_VEL
LIN {X 0,Y 362.529,Z 675.286,A -85,B 0,C 180,E1 -13062.882,E2 -13062.882} C_VEL
LIN {X 0,Y 363.366,Z 666.859,A -85,B 0,C 180,E1 -13064.277,E2 -13064.277} C_VEL
LIN {X 0,Y 364.393,Z 656.427,A -85,B 0,C 180,E1 -13065.665,E2 -13065.665} C_VEL
LIN {X 0,Y 365.396,Z 646.091,A -85,B 0,C 180,E1 -13066.769,E2 -13066.769} C_VEL
LIN {X 0,Y 366.408,Z 634.702,A -85,B 0,C 180,E1 -13067.728,E2 -13067.728} C_VEL
LIN {X 0,Y 367.558,Z 619.875,A -85,B 0,C 180,E1 -13068.68,E2 -13068.68} C_VEL
LIN {X 0,Y 368.966,Z 607.513,A -85,B 0,C 180,E1 -13069.472,E2 -13069.472} C_VEL
LIN {X 0,Y 370.209,Z 593.03,A -85,B 0,C 180,E1 -13070.162,E2 -13070.162} C_VEL
LIN {X 0,Y 371.099,Z 575.102,A -85,B 0,C 180,E1 -13070.727,E2 -13070.727} C_VEL
LIN {X 0,Y 373.372,Z 523.893,A -85,B 0,C 180,E1 -13072.218,E2 -13072.218} C_VEL
LIN {X 0,Y 372.106,Z 506.692,A -85,B 0,C 180,E1 -13072.952,E2 -13072.952} C_VEL
LIN {X 0,Y 369.531,Z 488.808,A -85,B 0,C 180,E1 -13073.892,E2 -13073.892} C_VEL
LIN {X 0,Y 366.613,Z 474.197,A -85,B 0,C 180,E1 -13074.826,E2 -13074.826} C_VEL
LIN {X 0,Y 369.011,Z 457.764,A -85,B 0,C 180,E1 -13078.434,E2 -13078.434} C_VEL
LIN {X 0,Y 368.189,Z 451.703,A -85,B 0,C 180,E1 -13080.053,E2 -13080.053} C_VEL
LIN {X 0,Y 366.127,Z 442.607,A -85,B 0,C 180,E1 -13082.839,E2 -13082.839} C_VEL
LIN {X 0,Y 364.136,Z 435.542,A -85,B 0,C 180,E1 -13085.381,E2 -13085.381} C_VEL
LIN {X 0,Y 362.616,Z 430.831,A -85,B 0,C 180,E1 -13087.379,E2 -13087.379} C_VEL
LIN {X 0,Y 361.882,Z 428.408,A -85,B 0,C 180,E1 -13088.573,E2 -13088.573} C_VEL
LIN {X 0,Y 361.837,Z 428.412,A -85,B 0,C 180,E1 -13092.432,E2 -13092.432} C_VEL
LIN {X 0,Y 361.82,Z 428.417,A -85,B 0,C 180,E1 -13095.947,E2 -13095.947} C_VEL
LIN {X 0,Y 361.838,Z 428.414,A -85,B 0,C 180,E1 -13099.245,E2 -13099.245} C_VEL
LIN {X 0,Y 361.866,Z 428.408,A -85,B 0,C 180,E1 -13102.777,E2 -13102.777} C_VEL
LIN {X 0,Y 361.856,Z 428.408,A -85,B 0,C 180,E1 -13105.72,E2 -13105.72} C_VEL
LIN {X 0,Y 361.875,Z 428.41,A -85,B 0,C 180,E1 -13109.672,E2 -13109.672} C_VEL
LIN {X 0,Y 361.962,Z 428.472,A -85,B 0,C 180,E1 -13113.709,E2 -13113.709} C_VEL
LIN {X 0,Y 362.448,Z 430.33,A -85,B 0,C 180,E1 -13114.749,E2 -13114.749} C_VEL
LIN {X 0,Y 367.319,Z 438.147,A -85,B 0,C 180,E1 -13115.767,E2 -13115.767} C_VEL
LIN {X 0,Y 373.433,Z 449.28,A -85,B 0,C 180,E1 -13116.982,E2 -13116.982} C_VEL
LIN {X 0,Y 376.003,Z 454.91,A -85,B 0,C 180,E1 -13117.501,E2 -13117.501} C_VEL
LIN {X 0,Y 372.128,Z 529.286,A -85,B 0,C 180,E1 -13119.73,E2 -13119.73} C_VEL
LIN {X 0,Y 371.544,Z 541.531,A -85,B 0,C 180,E1 -13120.238,E2 -13120.238} C_VEL
LIN {X 0,Y 370.826,Z 555.153,A -85,B 0,C 180,E1 -13121.061,E2 -13121.061} C_VEL
LIN {X 0,Y 369.825,Z 566.914,A -85,B 0,C 180,E1 -13121.984,E2 -13121.984} C_VEL
LIN {X 0,Y 368.626,Z 578.422,A -85,B 0,C 180,E1 -13123.145,E2 -13123.145} C_VEL
LIN {X 0,Y 367.408,Z 588.883,A -85,B 0,C 180,E1 -13124.467,E2 -13124.467} C_VEL
LIN {X 0,Y 366.101,Z 599.253,A -85,B 0,C 180,E1 -13126.116,E2 -13126.116} C_VEL
LIN {X 0,Y 364.92,Z 607.52,A -85,B 0,C 180,E1 -13127.769,E2 -13127.769} C_VEL
LIN {X 0,Y 363.889,Z 614.097,A -85,B 0,C 180,E1 -13129.428,E2 -13129.428} C_VEL
LIN {X 0,Y 363.066,Z 619.29,A -85,B 0,C 180,E1 -13131.091,E2 -13131.091} C_VEL
LIN {X 0,Y 362.345,Z 623.299,A -85,B 0,C 180,E1 -13132.757,E2 -13132.757} C_VEL
LIN {X 0,Y 361.935,Z 626.199,A -85,B 0,C 180,E1 -13134.428,E2 -13134.428} C_VEL
LIN {X 0,Y 361.616,Z 627.594,A -85,B 0,C 180,E1 -13135.541,E2 -13135.541} C_VEL
LIN {X 0,Y 361.272,Z 628.516,A -85,B 0,C 180,E1 -13136.654,E2 -13136.654} C_VEL
LIN {X 0,Y 361.02,Z 629.015,A -85,B 0,C 180,E1 -13137.769,E2 -13137.769} C_VEL
LIN {X 0,Y 360.888,Z 629.094,A -85,B 0,C 180,E1 -13138.884,E2 -13138.884} C_VEL
LIN {X 0,Y 360.838,Z 628.714,A -85,B 0,C 180,E1 -13140,E2 -13140} C_VEL
LIN {X 0,Y 360.868,Z 627.896,A -85,B 0,C 180,E1 -13141.116,E2 -13141.116} C_VEL
LIN {X 0,Y 360.949,Z 626.67,A -85,B 0,C 180,E1 -13142.232,E2 -13142.232} C_VEL
LIN {X 0,Y 361.154,Z 623.982,A -85,B 0,C 180,E1 -13143.905,E2 -13143.905} C_VEL
LIN {X 0,Y 361.279,Z 620.246,A -85,B 0,C 180,E1 -13145.582,E2 -13145.582} C_VEL
LIN {X 0,Y 361.518,Z 615.474,A -85,B 0,C 180,E1 -13147.215,E2 -13147.215} C_VEL
LIN {X 0,Y 361.864,Z 609.116,A -85,B 0,C 180,E1 -13148.939,E2 -13148.939} C_VEL
LIN {X 0,Y 362.449,Z 601.334,A -85,B 0,C 180,E1 -13150.615,E2 -13150.615} C_VEL
LIN {X 0,Y 362.936,Z 593.416,A -85,B 0,C 180,E1 -13152.015,E2 -13152.015} C_VEL
LIN {X 0,Y 363.594,Z 583.835,A -85,B 0,C 180,E1 -13153.412,E2 -13153.412} C_VEL
LIN {X 0,Y 364.302,Z 572.224,A -85,B 0,C 180,E1 -13154.771,E2 -13154.771} C_VEL
LIN {X 0,Y 364.952,Z 561.466,A -85,B 0,C 180,E1 -13155.784,E2 -13155.784} C_VEL
LIN {X 0,Y 365.466,Z 549.27,A -85,B 0,C 180,E1 -13156.694,E2 -13156.694} C_VEL
LIN {X 0,Y 365.997,Z 535.459,A -85,B 0,C 180,E1 -13157.46,E2 -13157.46} C_VEL
LIN {X 0,Y 366.35,Z 522.631,A -85,B 0,C 180,E1 -13157.947,E2 -13157.947} C_VEL
LIN {X 0,Y 368.025,Z 446.958,A -85,B 0,C 180,E1 -13159.877,E2 -13159.877} C_VEL
LIN {X 0,Y 361.923,Z 428.407,A -85,B 0,C 180,E1 -13160.646,E2 -13160.646} C_VEL
LIN {X 0,Y 361.895,Z 428.402,A -85,B 0,C 180,E1 -13164.113,E2 -13164.113} C_VEL
LIN {X 0,Y 361.943,Z 428.398,A -85,B 0,C 180,E1 -13166.721,E2 -13166.721} C_VEL
LIN {X 0,Y 361.875,Z 428.406,A -85,B 0,C 180,E1 -13170.328,E2 -13170.328} C_VEL
LIN {X 0,Y 361.857,Z 428.39,A -85,B 0,C 180,E1 -13174.28,E2 -13174.28} C_VEL
LIN {X 0,Y 361.866,Z 428.414,A -85,B 0,C 180,E1 -13177.223,E2 -13177.223} C_VEL
LIN {X 0,Y 361.837,Z 428.399,A -85,B 0,C 180,E1 -13180.755,E2 -13180.755} C_VEL
LIN {X 0,Y 361.82,Z 428.416,A -85,B 0,C 180,E1 -13184.368,E2 -13184.368} C_VEL
LIN {X 0,Y 361.838,Z 428.412,A -85,B 0,C 180,E1 -13187.568,E2 -13187.568} C_VEL
LIN {X 0,Y 361.871,Z 428.407,A -85,B 0,C 180,E1 -13190.973,E2 -13190.973} C_VEL
LIN {X 0,Y 361.876,Z 428.412,A -85,B 0,C 180,E1 -13194.655,E2 -13194.655} C_VEL
LIN {X 0,Y 361.84,Z 428.413,A -85,B 0,C 180,E1 -13198.371,E2 -13198.371} C_VEL
LIN {X 0,Y 361.901,Z 428.463,A -85,B 0,C 180,E1 -13199.446,E2 -13199.446} C_VEL
LIN {X 0,Y 365.042,Z 441.89,A -85,B 0,C 180,E1 -13202.328,E2 -13202.328} C_VEL
LIN {X 0,Y 366.984,Z 452.083,A -85,B 0,C 180,E1 -13204.433,E2 -13204.433} C_VEL
LIN {X 0,Y 366.113,Z 468.71,A -85,B 0,C 180,E1 -13207.423,E2 -13207.423} C_VEL
LIN {X 0,Y 365.963,Z 472.526,A -85,B 0,C 180,E1 -13208.065,E2 -13208.065} C_VEL
LIN {X 0,Y 370.446,Z 498.733,A -85,B 0,C 180,E1 -13208.891,E2 -13208.891} C_VEL
LIN {X 0,Y 369.045,Z 582.072,A -85,B 0,C 180,E1 -13210.533,E2 -13210.533} C_VEL
LIN {X 0,Y 368.591,Z 595.07,A -85,B 0,C 180,E1 -13210.978,E2 -13210.978} C_VEL
LIN {X 0,Y 367.925,Z 606.44,A -85,B 0,C 180,E1 -13211.556,E2 -13211.556} C_VEL
LIN {X 0,Y 366.964,Z 619.106,A -85,B 0,C 180,E1 -13212.444,E2 -13212.444} C_VEL
LIN {X 0,Y 365.931,Z 630.818,A -85,B 0,C 180,E1 -13213.519,E2 -13213.519} C_VEL
LIN {X 0,Y 365.047,Z 641.568,A -85,B 0,C 180,E1 -13214.793,E2 -13214.793} C_VEL
LIN {X 0,Y 363.811,Z 651.918,A -85,B 0,C 180,E1 -13216.312,E2 -13216.312} C_VEL
LIN {X 0,Y 362.899,Z 659.56,A -85,B 0,C 180,E1 -13217.7,E2 -13217.7} C_VEL
LIN {X 0,Y 362.091,Z 667.003,A -85,B 0,C 180,E1 -13219.374,E2 -13219.374} C_VEL
LIN {X 0,Y 361.394,Z 672.977,A -85,B 0,C 180,E1 -13221.05,E2 -13221.05} C_VEL
LIN {X 0,Y 360.996,Z 677.698,A -85,B 0,C 180,E1 -13222.73,E2 -13222.73} C_VEL
LIN {X 0,Y 360.716,Z 681.312,A -85,B 0,C 180,E1 -13224.409,E2 -13224.409} C_VEL
LIN {X 0,Y 360.543,Z 683.173,A -85,B 0,C 180,E1 -13225.528,E2 -13225.528} C_VEL
LIN {X 0,Y 360.4,Z 684.595,A -85,B 0,C 180,E1 -13226.646,E2 -13226.646} C_VEL
LIN {X 0,Y 360.35,Z 686.204,A -85,B 0,C 180,E1 -13228.882,E2 -13228.882} C_VEL
LIN {X 0,Y 360.344,Z 686.438,A -85,B 0,C 180,E1 -13230,E2 -13230} C_VEL
LIN {X 0,Y 360.35,Z 686.246,A -85,B 0,C 180,E1 -13231.118,E2 -13231.118} C_VEL
LIN {X 0,Y 360.399,Z 684.693,A -85,B 0,C 180,E1 -13233.354,E2 -13233.354} C_VEL
LIN {X 0,Y 360.541,Z 683.326,A -85,B 0,C 180,E1 -13234.472,E2 -13234.472} C_VEL
LIN {X 0,Y 360.774,Z 680.364,A -85,B 0,C 180,E1 -13236.195,E2 -13236.195} C_VEL
LIN {X 0,Y 360.95,Z 678.076,A -85,B 0,C 180,E1 -13237.216,E2 -13237.216} C_VEL
LIN {X 0,Y 360.472,Z 675.941,A -85,B 0,C 180,E1 -13238.089,E2 -13238.089} C_VEL
LIN {X 0,Y 358.012,Z 672.009,A -85,B 0,C 180,E1 -13239.49,E2 -13239.49} C_VEL
LIN {X 0,Y 355.71,Z 667.433,A -85,B 0,C 180,E1 -13240.855,E2 -13240.855} C_VEL
LIN {X 0,Y 355.482,Z 664.235,A -85,B 0,C 180,E1 -13241.658,E2 -13241.658} C_VEL
LIN {X 0,Y 356.448,Z 655.88,A -85,B 0,C 180,E1 -13243.396,E2 -13243.396} C_VEL
LIN {X 0,Y 357.542,Z 647.415,A -85,B 0,C 180,E1 -13244.805,E2 -13244.805} C_VEL
LIN {X 0,Y 358.548,Z 637.449,A -85,B 0,C 180,E1 -13246.164,E2 -13246.164} C_VEL
LIN {X 0,Y 359.611,Z 626.691,A -85,B 0,C 180,E1 -13247.34,E2 -13247.34} C_VEL
LIN {X 0,Y 360.586,Z 615.211,A -85,B 0,C 180,E1 -13248.318,E2 -13248.318} C_VEL
LIN {X 0,Y 361.537,Z 602.23,A -85,B 0,C 180,E1 -13249.15,E2 -13249.15} C_VEL
LIN {X 0,Y 362.097,Z 589.855,A -85,B 0,C 180,E1 -13249.709,E2 -13249.709} C_VEL
LIN {X 0,Y 362.626,Z 575.803,A -85,B 0,C 180,E1 -13250.085,E2 -13250.085} C_VEL
LIN {X 0,Y 363.804,Z 498.418,A -85,B 0,C 180,E1 -13251.626,E2 -13251.626} C_VEL
LIN {X 0,Y 359.181,Z 472.722,A -85,B 0,C 180,E1 -13252.467,E2 -13252.467} C_VEL
LIN {X 0,Y 360.105,Z 456.128,A -85,B 0,C 180,E1 -13255.427,E2 -13255.427} C_VEL
LIN {X 0,Y 360.059,Z 452.527,A -85,B 0,C 180,E1 -13256.119,E2 -13256.119} C_VEL
LIN {X 0,Y 357.452,Z 439.913,A -85,B 0,C 180,E1 -13258.797,E2 -13258.797} C_VEL
LIN {X 0,Y 354.837,Z 429.286,A -85,B 0,C 180,E1 -13261.159,E2 -13261.159} C_VEL
LIN {X 0,Y 354.814,Z 429.289,A -85,B 0,C 180,E1 -13265.059,E2 -13265.059} C_VEL
LIN {X 0,Y 354.807,Z 429.287,A -85,B 0,C 180,E1 -13267.883,E2 -13267.883} C_VEL
LIN {X 0,Y 354.79,Z 429.289,A -85,B 0,C 180,E1 -13271.172,E2 -13271.172} C_VEL
LIN {X 0,Y 354.791,Z 429.285,A -85,B 0,C 180,E1 -13274.511,E2 -13274.511} C_VEL
LIN {X 0,Y 354.797,Z 429.282,A -85,B 0,C 180,E1 -13277.663,E2 -13277.663} C_VEL
LIN {X 0,Y 354.817,Z 429.291,A -85,B 0,C 180,E1 -13280.666,E2 -13280.666} C_VEL
LIN {X 0,Y 354.824,Z 429.272,A -85,B 0,C 180,E1 -13284.301,E2 -13284.301} C_VEL
LIN {X 0,Y 354.789,Z 429.29,A -85,B 0,C 180,E1 -13287.667,E2 -13287.667} C_VEL
LIN {X 0,Y 354.862,Z 429.399,A -85,B 0,C 180,E1 -13290.378,E2 -13290.378} C_VEL
LIN {X 0,Y 358.037,Z 444.548,A -85,B 0,C 180,E1 -13293.471,E2 -13293.471} C_VEL
LIN {X 0,Y 359.11,Z 451.251,A -85,B 0,C 180,E1 -13294.807,E2 -13294.807} C_VEL
LIN {X 0,Y 358.198,Z 466.451,A -85,B 0,C 180,E1 -13297.633,E2 -13297.633} C_VEL
LIN {X 0,Y 357.885,Z 473.402,A -85,B 0,C 180,E1 -13298.905,E2 -13298.905} C_VEL
LIN {X 0,Y 361.197,Z 498.931,A -85,B 0,C 180,E1 -13299.743,E2 -13299.743} C_VEL
LIN {X 0,Y 359.027,Z 584.807,A -85,B 0,C 180,E1 -13302.006,E2 -13302.006} C_VEL
LIN {X 0,Y 358.483,Z 598.519,A -85,B 0,C 180,E1 -13302.604,E2 -13302.604} C_VEL
LIN {X 0,Y 357.913,Z 610.13,A -85,B 0,C 180,E1 -13303.311,E2 -13303.311} C_VEL
LIN {X 0,Y 357.18,Z 622.335,A -85,B 0,C 180,E1 -13304.282,E2 -13304.282} C_VEL
LIN {X 0,Y 356.479,Z 633.817,A -85,B 0,C 180,E1 -13305.441,E2 -13305.441} C_VEL
LIN {X 0,Y 355.685,Z 645.06,A -85,B 0,C 180,E1 -13306.866,E2 -13306.866} C_VEL
LIN {X 0,Y 354.97,Z 654.155,A -85,B 0,C 180,E1 -13308.291,E2 -13308.291} C_VEL
LIN {X 0,Y 354.332,Z 663.02,A -85,B 0,C 180,E1 -13310.006,E2 -13310.006} C_VEL
LIN {X 0,Y 353.843,Z 670.109,A -85,B 0,C 180,E1 -13311.721,E2 -13311.721} C_VEL
LIN {X 0,Y 353.528,Z 676.537,A -85,B 0,C 180,E1 -13313.712,E2 -13313.712} C_VEL
LIN {X 0,Y 353.412,Z 680.727,A -85,B 0,C 180,E1 -13315.438,E2 -13315.438} C_VEL
LIN {X 0,Y 353.291,Z 682.839,A -85,B 0,C 180,E1 -13316.579,E2 -13316.579} C_VEL
LIN {X 0,Y 353.227,Z 684.514,A -85,B 0,C 180,E1 -13317.719,E2 -13317.719} C_VEL
LIN {X 0,Y 353.213,Z 685.731,A -85,B 0,C 180,E1 -13318.86,E2 -13318.86} C_VEL
LIN {X 0,Y 353.243,Z 686.483,A -85,B 0,C 180,E1 -13320,E2 -13320} C_VEL
LIN {X 0,Y 353.274,Z 686.826,A -85,B 0,C 180,E1 -13321.14,E2 -13321.14} C_VEL
LIN {X 0,Y 353.322,Z 686.712,A -85,B 0,C 180,E1 -13322.28,E2 -13322.28} C_VEL
LIN {X 0,Y 353.363,Z 686.151,A -85,B 0,C 180,E1 -13323.421,E2 -13323.421} C_VEL
LIN {X 0,Y 353.5,Z 685.175,A -85,B 0,C 180,E1 -13324.561,E2 -13324.561} C_VEL
LIN {X 0,Y 353.787,Z 683.724,A -85,B 0,C 180,E1 -13325.7,E2 -13325.7} C_VEL
LIN {X 0,Y 354.081,Z 680.705,A -85,B 0,C 180,E1 -13327.412,E2 -13327.412} C_VEL
LIN {X 0,Y 354.636,Z 676.594,A -85,B 0,C 180,E1 -13329.122,E2 -13329.122} C_VEL
LIN {X 0,Y 355.532,Z 670.276,A -85,B 0,C 180,E1 -13331.112,E2 -13331.112} C_VEL
LIN {X 0,Y 356.566,Z 663.276,A -85,B 0,C 180,E1 -13332.811,E2 -13332.811} C_VEL
LIN {X 0,Y 357.743,Z 654.596,A -85,B 0,C 180,E1 -13334.506,E2 -13334.506} C_VEL
LIN {X 0,Y 359.154,Z 644.701,A -85,B 0,C 180,E1 -13336.051,E2 -13336.051} C_VEL
LIN {X 0,Y 360.58,Z 633.657,A -85,B 0,C 180,E1 -13337.438,E2 -13337.438} C_VEL
LIN {X 0,Y 361.999,Z 621.067,A -85,B 0,C 180,E1 -13338.683,E2 -13338.683} C_VEL
LIN {X 0,Y 363.221,Z 608.372,A -85,B 0,C 180,E1 -13339.645,E2 -13339.645} C_VEL
LIN {X 0,Y 364.289,Z 595.333,A -85,B 0,C 180,E1 -13340.394,E2 -13340.394} C_VEL
LIN {X 0,Y 365.217,Z 581.78,A -85,B 0,C 180,E1 -13340.929,E2 -13340.929} C_VEL
LIN {X 0,Y 369.156,Z 508.889,A -85,B 0,C 180,E1 -13343.125,E2 -13343.125} C_VEL
LIN {X 0,Y 369.464,Z 500.646,A -85,B 0,C 180,E1 -13343.407,E2 -13343.407} C_VEL
LIN {X 0,Y 367.039,Z 487.409,A -85,B 0,C 180,E1 -13344.211,E2 -13344.211} C_VEL
LIN {X 0,Y 364.266,Z 475.762,A -85,B 0,C 180,E1 -13345.074,E2 -13345.074} C_VEL
LIN {X 0,Y 365.476,Z 464.642,A -85,B 0,C 180,E1 -13347.277,E2 -13347.277} C_VEL
LIN {X 0,Y 364.574,Z 458.29,A -85,B 0,C 180,E1 -13348.812,E2 -13348.812} C_VEL
LIN {X 0,Y 362.822,Z 450.886,A -85,B 0,C 180,E1 -13350.824,E2 -13350.824} C_VEL
LIN {X 0,Y 360.068,Z 442.022,A -85,B 0,C 180,E1 -13353.584,E2 -13353.584} C_VEL
LIN {X 0,Y 358.085,Z 436.819,A -85,B 0,C 180,E1 -13355.462,E2 -13355.462} C_VEL
LIN {X 0,Y 356.484,Z 433.036,A -85,B 0,C 180,E1 -13357.018,E2 -13357.018} C_VEL
LIN {X 0,Y 355.49,Z 431.527,A -85,B 0,C 180,E1 -13357.797,E2 -13357.797} C_VEL
LIN {X 0,Y 354.833,Z 429.287,A -85,B 0,C 180,E1 -13358.784,E2 -13358.784} C_VEL
LIN {X 0,Y 354.796,Z 429.292,A -85,B 0,C 180,E1 -13362.337,E2 -13362.337} C_VEL
LIN {X 0,Y 354.769,Z 429.296,A -85,B 0,C 180,E1 -13366.104,E2 -13366.104} C_VEL
LIN {X 0,Y 354.79,Z 429.288,A -85,B 0,C 180,E1 -13369.179,E2 -13369.179} C_VEL
LIN {X 0,Y 354.809,Z 429.285,A -85,B 0,C 180,E1 -13372.403,E2 -13372.403} C_VEL
LIN {X 0,Y 354.825,Z 429.284,A -85,B 0,C 180,E1 -13375.976,E2 -13375.976} C_VEL
LIN {X 0,Y 354.857,Z 429.557,A -85,B 0,C 180,E1 -13376.286,E2 -13376.286} C_VEL
LIN {X 0,Y 355.66,Z 431.875,A -85,B 0,C 180,E1 -13377.084,E2 -13377.084} C_VEL
LIN {X 0,Y 356.311,Z 432.829,A -85,B 0,C 180,E1 -13377.487,E2 -13377.487} C_VEL
LIN {X 0,Y 357.258,Z 437.278,A -85,B 0,C 180,E1 -13378.576,E2 -13378.576} C_VEL
LIN {X 0,Y 359.664,Z 447.877,A -85,B 0,C 180,E1 -13380.757,E2 -13380.757} C_VEL
LIN {X 0,Y 361.229,Z 453.518,A -85,B 0,C 180,E1 -13381.783,E2 -13381.783} C_VEL
LIN {X 0,Y 361.915,Z 466.118,A -85,B 0,C 180,E1 -13383.288,E2 -13383.288} C_VEL
LIN {X 0,Y 362.9,Z 480.637,A -85,B 0,C 180,E1 -13384.782,E2 -13384.782} C_VEL
LIN {X 0,Y 363.381,Z 485.337,A -85,B 0,C 180,E1 -13385.178,E2 -13385.178} C_VEL
LIN {X 0,Y 365.842,Z 502.387,A -85,B 0,C 180,E1 -13386.208,E2 -13386.208} C_VEL
LIN {X 0,Y 366.861,Z 514.535,A -85,B 0,C 180,E1 -13386.808,E2 -13386.808} C_VEL
LIN {X 0,Y 367.45,Z 527.977,A -85,B 0,C 180,E1 -13387.396,E2 -13387.396} C_VEL
LIN {X 0,Y 363.713,Z 596.04,A -85,B 0,C 180,E1 -13389.499,E2 -13389.499} C_VEL
LIN {X 0,Y 362.818,Z 610.628,A -85,B 0,C 180,E1 -13390,E2 -13390} C_VEL
LIN {X 0,Y 361.728,Z 624.276,A -85,B 0,C 180,E1 -13390.713,E2 -13390.713} C_VEL
LIN {X 0,Y 360.599,Z 636.016,A -85,B 0,C 180,E1 -13391.536,E2 -13391.536} C_VEL
LIN {X 0,Y 359.398,Z 646.822,A -85,B 0,C 180,E1 -13392.503,E2 -13392.503} C_VEL
LIN {X 0,Y 358.141,Z 658.022,A -85,B 0,C 180,E1 -13393.761,E2 -13393.761} C_VEL
LIN {X 0,Y 356.91,Z 668.03,A -85,B 0,C 180,E1 -13395.168,E2 -13395.168} C_VEL
LIN {X 0,Y 355.912,Z 676.338,A -85,B 0,C 180,E1 -13396.584,E2 -13396.584} C_VEL
LIN {X 0,Y 354.931,Z 684.457,A -85,B 0,C 180,E1 -13398.29,E2 -13398.29} C_VEL
LIN {X 0,Y 354.181,Z 691.864,A -85,B 0,C 180,E1 -13400.29,E2 -13400.29} C_VEL
LIN {X 0,Y 353.661,Z 696.791,A -85,B 0,C 180,E1 -13402.004,E2 -13402.004} C_VEL
LIN {X 0,Y 353.389,Z 700.852,A -85,B 0,C 180,E1 -13403.919,E2 -13403.919} C_VEL
LIN {X 0,Y 353.345,Z 703.131,A -85,B 0,C 180,E1 -13405.437,E2 -13405.437} C_VEL
LIN {X 0,Y 353.284,Z 704.274,A -85,B 0,C 180,E1 -13406.579,E2 -13406.579} C_VEL
LIN {X 0,Y 353.235,Z 704.99,A -85,B 0,C 180,E1 -13407.719,E2 -13407.719} C_VEL
LIN {X 0,Y 353.336,Z 705.448,A -85,B 0,C 180,E1 -13410,E2 -13410} C_VEL
LIN {X 0,Y 353.276,Z 705.223,A -85,B 0,C 180,E1 -13411.14,E2 -13411.14} C_VEL
LIN {X 0,Y 353.285,Z 703.594,A -85,B 0,C 180,E1 -13413.421,E2 -13413.421} C_VEL
LIN {X 0,Y 353.327,Z 702.159,A -85,B 0,C 180,E1 -13414.564,E2 -13414.564} C_VEL
LIN {X 0,Y 353.388,Z 699.567,A -85,B 0,C 180,E1 -13416.079,E2 -13416.079} C_VEL
LIN {X 0,Y 353.638,Z 695.125,A -85,B 0,C 180,E1 -13417.997,E2 -13417.997} C_VEL
LIN {X 0,Y 354.153,Z 688.882,A -85,B 0,C 180,E1 -13420,E2 -13420} C_VEL
LIN {X 0,Y 354.797,Z 682.069,A -85,B 0,C 180,E1 -13421.715,E2 -13421.715} C_VEL
LIN {X 0,Y 355.579,Z 675.099,A -85,B 0,C 180,E1 -13423.138,E2 -13423.138} C_VEL
LIN {X 0,Y 356.478,Z 666.674,A -85,B 0,C 180,E1 -13424.559,E2 -13424.559} C_VEL
LIN {X 0,Y 357.532,Z 656.244,A -85,B 0,C 180,E1 -13425.974,E2 -13425.974} C_VEL
LIN {X 0,Y 358.599,Z 645.912,A -85,B 0,C 180,E1 -13427.096,E2 -13427.096} C_VEL
LIN {X 0,Y 359.657,Z 634.529,A -85,B 0,C 180,E1 -13428.072,E2 -13428.072} C_VEL
LIN {X 0,Y 360.691,Z 622.769,A -85,B 0,C 180,E1 -13428.901,E2 -13428.901} C_VEL
LIN {X 0,Y 362.337,Z 609.411,A -85,B 0,C 180,E1 -13429.843,E2 -13429.843} C_VEL
LIN {X 0,Y 363.678,Z 595.378,A -85,B 0,C 180,E1 -13430.577,E2 -13430.577} C_VEL
LIN {X 0,Y 364.728,Z 580.628,A -85,B 0,C 180,E1 -13431.106,E2 -13431.106} C_VEL
LIN {X 0,Y 367.367,Z 524.958,A -85,B 0,C 180,E1 -13432.78,E2 -13432.78} C_VEL
LIN {X 0,Y 366.29,Z 508.907,A -85,B 0,C 180,E1 -13433.491,E2 -13433.491} C_VEL
LIN {X 0,Y 364.12,Z 492.637,A -85,B 0,C 180,E1 -13434.372,E2 -13434.372} C_VEL
LIN {X 0,Y 360.854,Z 476.099,A -85,B 0,C 180,E1 -13435.461,E2 -13435.461} C_VEL
LIN {X 0,Y 360.253,Z 472.944,A -85,B 0,C 180,E1 -13435.707,E2 -13435.707} C_VEL
LIN {X 0,Y 362.387,Z 459.792,A -85,B 0,C 180,E1 -13438.685,E2 -13438.685} C_VEL
LIN {X 0,Y 361.577,Z 453.787,A -85,B 0,C 180,E1 -13440.356,E2 -13440.356} C_VEL
LIN {X 0,Y 359.564,Z 444.92,A -85,B 0,C 180,E1 -13443.181,E2 -13443.181} C_VEL
LIN {X 0,Y 357.334,Z 436.912,A -85,B 0,C 180,E1 -13446.256,E2 -13446.256} C_VEL
LIN {X 0,Y 355.753,Z 432.189,A -85,B 0,C 180,E1 -13448.483,E2 -13448.483} C_VEL
LIN {X 0,Y 354.794,Z 429.292,A -85,B 0,C 180,E1 -13450.167,E2 -13450.167} C_VEL
LIN {X 0,Y 354.769,Z 429.293,A -85,B 0,C 180,E1 -13453.896,E2 -13453.896} C_VEL
LIN {X 0,Y 354.796,Z 429.291,A -85,B 0,C 180,E1 -13457.663,E2 -13457.663} C_VEL
LIN {X 0,Y 354.817,Z 429.289,A -85,B 0,C 180,E1 -13460.666,E2 -13460.666} C_VEL
LIN {X 0,Y 354.824,Z 429.284,A -85,B 0,C 180,E1 -13464.301,E2 -13464.301} C_VEL
LIN {X 0,Y 354.789,Z 429.291,A -85,B 0,C 180,E1 -13467.667,E2 -13467.667} C_VEL
LIN {X 0,Y 354.849,Z 429.285,A -85,B 0,C 180,E1 -13471.619,E2 -13471.619} C_VEL
LIN {X 0,Y 354.922,Z 429.505,A -85,B 0,C 180,E1 -13472.268,E2 -13472.268} C_VEL
LIN {X 0,Y 355.702,Z 431.907,A -85,B 0,C 180,E1 -13473.762,E2 -13473.762} C_VEL
LIN {X 0,Y 357.892,Z 435.281,A -85,B 0,C 180,E1 -13474.272,E2 -13474.272} C_VEL
LIN {X 0,Y 362.667,Z 442.687,A -85,B 0,C 180,E1 -13475.32,E2 -13475.32} C_VEL
LIN {X 0,Y 368.52,Z 453.606,A -85,B 0,C 180,E1 -13476.562,E2 -13476.562} C_VEL
LIN {X 0,Y 370.133,Z 457.115,A -85,B 0,C 180,E1 -13476.895,E2 -13476.895} C_VEL
LIN {X 0,Y 366.425,Z 520.141,A -85,B 0,C 180,E1 -13478.849,E2 -13478.849} C_VEL
LIN {X 0,Y 365.695,Z 537.652,A -85,B 0,C 180,E1 -13479.468,E2 -13479.468} C_VEL
LIN {X 0,Y 364.984,Z 550.382,A -85,B 0,C 180,E1 -13480.161,E2 -13480.161} C_VEL
LIN {X 0,Y 363.954,Z 563.506,A -85,B 0,C 180,E1 -13481.12,E2 -13481.12} C_VEL
LIN {X 0,Y 362.722,Z 575.347,A -85,B 0,C 180,E1 -13482.236,E2 -13482.236} C_VEL
LIN {X 0,Y 361.409,Z 585.906,A -85,B 0,C 180,E1 -13483.477,E2 -13483.477} C_VEL
LIN {X 0,Y 360.08,Z 596.202,A -85,B 0,C 180,E1 -13485.012,E2 -13485.012} C_VEL
LIN {X 0,Y 358.981,Z 603.832,A -85,B 0,C 180,E1 -13486.412,E2 -13486.412} C_VEL
LIN {X 0,Y 357.759,Z 611.317,A -85,B 0,C 180,E1 -13488.096,E2 -13488.096} C_VEL
LIN {X 0,Y 356.806,Z 617.272,A -85,B 0,C 180,E1 -13489.789,E2 -13489.789} C_VEL
LIN {X 0,Y 355.962,Z 621.942,A -85,B 0,C 180,E1 -13491.484,E2 -13491.484} C_VEL
LIN {X 0,Y 355.245,Z 625.461,A -85,B 0,C 180,E1 -13493.183,E2 -13493.183} C_VEL
LIN {X 0,Y 354.94,Z 627.214,A -85,B 0,C 180,E1 -13494.318,E2 -13494.318} C_VEL
LIN {X 0,Y 354.6,Z 628.511,A -85,B 0,C 180,E1 -13495.453,E2 -13495.453} C_VEL
LIN {X 0,Y 354.243,Z 629.373,A -85,B 0,C 180,E1 -13496.588,E2 -13496.588} C_VEL
LIN {X 0,Y 353.981,Z 629.822,A -85,B 0,C 180,E1 -13497.724,E2 -13497.724} C_VEL
LIN {X 0,Y 353.84,Z 629.833,A -85,B 0,C 180,E1 -13498.862,E2 -13498.862} C_VEL
LIN {X 0,Y 353.789,Z 629.374,A -85,B 0,C 180,E1 -13500,E2 -13500} C_VEL
LIN {X 0,Y 353.821,Z 628.498,A -85,B 0,C 180,E1 -13501.138,E2 -13501.138} C_VEL
LIN {X 0,Y 353.879,Z 627.209,A -85,B 0,C 180,E1 -13502.276,E2 -13502.276} C_VEL
LIN {X 0,Y 354.102,Z 624.407,A -85,B 0,C 180,E1 -13503.983,E2 -13503.983} C_VEL
LIN {X 0,Y 354.212,Z 620.55,A -85,B 0,C 180,E1 -13505.694,E2 -13505.694} C_VEL
LIN {X 0,Y 354.531,Z 614.769,A -85,B 0,C 180,E1 -13507.618,E2 -13507.618} C_VEL
LIN {X 0,Y 354.91,Z 607.927,A -85,B 0,C 180,E1 -13509.403,E2 -13509.403} C_VEL
LIN {X 0,Y 355.516,Z 599.697,A -85,B 0,C 180,E1 -13511.113,E2 -13511.113} C_VEL
LIN {X 0,Y 356.228,Z 589.417,A -85,B 0,C 180,E1 -13512.824,E2 -13512.824} C_VEL
LIN {X 0,Y 356.97,Z 578.687,A -85,B 0,C 180,E1 -13514.247,E2 -13514.247} C_VEL
LIN {X 0,Y 357.694,Z 566.64,A -85,B 0,C 180,E1 -13515.529,E2 -13515.529} C_VEL
LIN {X 0,Y 358.212,Z 554.696,A -85,B 0,C 180,E1 -13516.528,E2 -13516.528} C_VEL
LIN {X 0,Y 358.824,Z 541.359,A -85,B 0,C 180,E1 -13517.379,E2 -13517.379} C_VEL
LIN {X 0,Y 359.235,Z 527.98,A -85,B 0,C 180,E1 -13517.984,E2 -13517.984} C_VEL
LIN {X 0,Y 359.684,Z 506.541,A -85,B 0,C 180,E1 -13518.587,E2 -13518.587} C_VEL
LIN {X 0,Y 361.105,Z 448.415,A -85,B 0,C 180,E1 -13520.104,E2 -13520.104} C_VEL
LIN {X 0,Y 354.85,Z 429.289,A -85,B 0,C 180,E1 -13520.925,E2 -13520.925} C_VEL
LIN {X 0,Y 354.862,Z 429.278,A -85,B 0,C 180,E1 -13524.576,E2 -13524.576} C_VEL
LIN {X 0,Y 354.884,Z 429.276,A -85,B 0,C 180,E1 -13527.096,E2 -13527.096} C_VEL
LIN {X 0,Y 354.802,Z 429.288,A -85,B 0,C 180,E1 -13530.999,E2 -13530.999} C_VEL
LIN {X 0,Y 354.808,Z 429.264,A -85,B 0,C 180,E1 -13533.702,E2 -13533.702} C_VEL
LIN {X 0,Y 354.8,Z 429.288,A -85,B 0,C 180,E1 -13536.459,E2 -13536.459} C_VEL
LIN {X 0,Y 354.826,Z 429.276,A -85,B 0,C 180,E1 -13539.424,E2 -13539.424} C_VEL
LIN {X 0,Y 354.79,Z 429.294,A -85,B 0,C 180,E1 -13542.867,E2 -13542.867} C_VEL
LIN {X 0,Y 354.769,Z 429.28,A -85,B 0,C 180,E1 -13546.104,E2 -13546.104} C_VEL
LIN {X 0,Y 354.79,Z 429.284,A -85,B 0,C 180,E1 -13549.179,E2 -13549.179} C_VEL
LIN {X 0,Y 354.809,Z 429.287,A -85,B 0,C 180,E1 -13552.403,E2 -13552.403} C_VEL
LIN {X 0,Y 354.814,Z 429.289,A -85,B 0,C 180,E1 -13554.941,E2 -13554.941} C_VEL
LIN {X 0,Y 354.843,Z 429.405,A -85,B 0,C 180,E1 -13559.005,E2 -13559.005} C_VEL
LIN {X 0,Y 357.634,Z 440.878,A -85,B 0,C 180,E1 -13561.54,E2 -13561.54} C_VEL
LIN {X 0,Y 360.177,Z 453.313,A -85,B 0,C 180,E1 -13564.16,E2 -13564.16} C_VEL
LIN {X 0,Y 359.454,Z 466.615,A -85,B 0,C 180,E1 -13566.585,E2 -13566.585} C_VEL
LIN {X 0,Y 359.256,Z 472.901,A -85,B 0,C 180,E1 -13567.648,E2 -13567.648} C_VEL
LIN {X 0,Y 363.769,Z 498.353,A -85,B 0,C 180,E1 -13568.474,E2 -13568.474} C_VEL
LIN {X 0,Y 362.527,Z 577.881,A -85,B 0,C 180,E1 -13570.058,E2 -13570.058} C_VEL
LIN {X 0,Y 362.082,Z 591.024,A -85,B 0,C 180,E1 -13570.438,E2 -13570.438} C_VEL
LIN {X 0,Y 361.317,Z 604.174,A -85,B 0,C 180,E1 -13571.059,E2 -13571.059} C_VEL
LIN {X 0,Y 360.484,Z 615.769,A -85,B 0,C 180,E1 -13571.824,E2 -13571.824} C_VEL
LIN {X 0,Y 359.525,Z 627.112,A -85,B 0,C 180,E1 -13572.803,E2 -13572.803} C_VEL
LIN {X 0,Y 358.581,Z 637.145,A -85,B 0,C 180,E1 -13573.902,E2 -13573.902} C_VEL
LIN {X 0,Y 357.621,Z 646.734,A -85,B 0,C 180,E1 -13575.198,E2 -13575.198} C_VEL
LIN {X 0,Y 356.464,Z 655.319,A -85,B 0,C 180,E1 -13576.605,E2 -13576.605} C_VEL
LIN {X 0,Y 355.527,Z 663.675,A -85,B 0,C 180,E1 -13578.31,E2 -13578.31} C_VEL
LIN {X 0,Y 354.892,Z 669.357,A -85,B 0,C 180,E1 -13579.733,E2 -13579.733} C_VEL
LIN {X 0,Y 354.2,Z 674.886,A -85,B 0,C 180,E1 -13581.442,E2 -13581.442} C_VEL
LIN {X 0,Y 353.794,Z 679.599,A -85,B 0,C 180,E1 -13583.334,E2 -13583.334} C_VEL
LIN {X 0,Y 353.482,Z 683.362,A -85,B 0,C 180,E1 -13585.438,E2 -13585.438} C_VEL
LIN {X 0,Y 353.322,Z 684.784,A -85,B 0,C 180,E1 -13586.579,E2 -13586.579} C_VEL
LIN {X 0,Y 353.252,Z 686.393,A -85,B 0,C 180,E1 -13588.86,E2 -13588.86} C_VEL
LIN {X 0,Y 353.248,Z 686.627,A -85,B 0,C 180,E1 -13590,E2 -13590} C_VEL
LIN {X 0,Y 353.252,Z 686.435,A -85,B 0,C 180,E1 -13591.14,E2 -13591.14} C_VEL
LIN {X 0,Y 353.321,Z 684.881,A -85,B 0,C 180,E1 -13593.421,E2 -13593.421} C_VEL
LIN {X 0,Y 353.48,Z 683.513,A -85,B 0,C 180,E1 -13594.562,E2 -13594.562} C_VEL
LIN {X 0,Y 353.786,Z 679.838,A -85,B 0,C 180,E1 -13596.655,E2 -13596.655} C_VEL
LIN {X 0,Y 354.199,Z 675.166,A -85,B 0,C 180,E1 -13598.558,E2 -13598.558} C_VEL
LIN {X 0,Y 354.858,Z 669.706,A -85,B 0,C 180,E1 -13600.268,E2 -13600.268} C_VEL
LIN {X 0,Y 355.482,Z 664.235,A -85,B 0,C 180,E1 -13601.658,E2 -13601.658} C_VEL
LIN {X 0,Y 355.296,Z 660.863,A -85,B 0,C 180,E1 -13602.439,E2 -13602.439} C_VEL
LIN {X 0,Y 353.238,Z 655.063,A -85,B 0,C 180,E1 -13603.698,E2 -13603.698} C_VEL
LIN {X 0,Y 351.214,Z 648.747,A -85,B 0,C 180,E1 -13604.894,E2 -13604.894} C_VEL
LIN {X 0,Y 351.076,Z 644.469,A -85,B 0,C 180,E1 -13605.566,E2 -13605.566} C_VEL
LIN {X 0,Y 352.079,Z 633.926,A -85,B 0,C 180,E1 -13606.929,E2 -13606.929} C_VEL
LIN {X 0,Y 353.284,Z 622.304,A -85,B 0,C 180,E1 -13608.11,E2 -13608.11} C_VEL
LIN {X 0,Y 354.267,Z 610.441,A -85,B 0,C 180,E1 -13609.032,E2 -13609.032} C_VEL
LIN {X 0,Y 355.106,Z 597.519,A -85,B 0,C 180,E1 -13609.774,E2 -13609.774} C_VEL
LIN {X 0,Y 355.592,Z 585.872,A -85,B 0,C 180,E1 -13610.235,E2 -13610.235} C_VEL
LIN {X 0,Y 356.248,Z 559.838,A -85,B 0,C 180,E1 -13610.8,E2 -13610.8} C_VEL
LIN {X 0,Y 357.207,Z 499.378,A -85,B 0,C 180,E1 -13612.027,E2 -13612.027} C_VEL
LIN {X 0,Y 352.476,Z 472.799,A -85,B 0,C 180,E1 -13612.923,E2 -13612.923} C_VEL
LIN {X 0,Y 353.429,Z 456.157,A -85,B 0,C 180,E1 -13615.943,E2 -13615.943} C_VEL
LIN {X 0,Y 352.05,Z 448.224,A -85,B 0,C 180,E1 -13617.574,E2 -13617.574} C_VEL
LIN {X 0,Y 349.367,Z 436.415,A -85,B 0,C 180,E1 -13620.193,E2 -13620.193} C_VEL
LIN {X 0,Y 347.773,Z 430.168,A -85,B 0,C 180,E1 -13621.612,E2 -13621.612} C_VEL
LIN {X 0,Y 347.746,Z 430.172,A -85,B 0,C 180,E1 -13624.464,E2 -13624.464} C_VEL
LIN {X 0,Y 347.775,Z 430.164,A -85,B 0,C 180,E1 -13627.989,E2 -13627.989} C_VEL
LIN {X 0,Y 347.753,Z 430.169,A -85,B 0,C 180,E1 -13631.83,E2 -13631.83} C_VEL
LIN {X 0,Y 347.769,Z 430.165,A -85,B 0,C 180,E1 -13635.017,E2 -13635.017} C_VEL
LIN {X 0,Y 347.753,Z 430.157,A -85,B 0,C 180,E1 -13638.397,E2 -13638.397} C_VEL
LIN {X 0,Y 347.776,Z 430.163,A -85,B 0,C 180,E1 -13642.011,E2 -13642.011} C_VEL
LIN {X 0,Y 347.747,Z 430.165,A -85,B 0,C 180,E1 -13645.536,E2 -13645.536} C_VEL
LIN {X 0,Y 347.762,Z 430.167,A -85,B 0,C 180,E1 -13649.653,E2 -13649.653} C_VEL
LIN {X 0,Y 347.819,Z 430.278,A -85,B 0,C 180,E1 -13650.121,E2 -13650.121} C_VEL
LIN {X 0,Y 350.971,Z 445.266,A -85,B 0,C 180,E1 -13653.221,E2 -13653.221} C_VEL
LIN {X 0,Y 352.135,Z 452.05,A -85,B 0,C 180,E1 -13654.589,E2 -13654.589} C_VEL
LIN {X 0,Y 351.305,Z 466.365,A -85,B 0,C 180,E1 -13657.292,E2 -13657.292} C_VEL
LIN {X 0,Y 350.945,Z 473.706,A -85,B 0,C 180,E1 -13658.621,E2 -13658.621} C_VEL
LIN {X 0,Y 354.298,Z 499.658,A -85,B 0,C 180,E1 -13659.497,E2 -13659.497} C_VEL
LIN {X 0,Y 352.055,Z 584.438,A -85,B 0,C 180,E1 -13661.787,E2 -13661.787} C_VEL
LIN {X 0,Y 351.498,Z 598.26,A -85,B 0,C 180,E1 -13662.397,E2 -13662.397} C_VEL
LIN {X 0,Y 350.924,Z 609.985,A -85,B 0,C 180,E1 -13663.118,E2 -13663.118} C_VEL
LIN {X 0,Y 350.156,Z 622.452,A -85,B 0,C 180,E1 -13664.13,E2 -13664.13} C_VEL
LIN {X 0,Y 349.453,Z 633.755,A -85,B 0,C 180,E1 -13665.291,E2 -13665.291} C_VEL
LIN {X 0,Y 348.638,Z 645.023,A -85,B 0,C 180,E1 -13666.744,E2 -13666.744} C_VEL
LIN {X 0,Y 347.949,Z 653.339,A -85,B 0,C 180,E1 -13668.051,E2 -13668.051} C_VEL
LIN {X 0,Y 347.309,Z 662.376,A -85,B 0,C 180,E1 -13669.801,E2 -13669.801} C_VEL
LIN {X 0,Y 346.804,Z 669.663,A -85,B 0,C 180,E1 -13671.551,E2 -13671.551} C_VEL
LIN {X 0,Y 346.486,Z 675.671,A -85,B 0,C 180,E1 -13673.391,E2 -13673.391} C_VEL
LIN {X 0,Y 346.329,Z 680.547,A -85,B 0,C 180,E1 -13675.344,E2 -13675.344} C_VEL
LIN {X 0,Y 346.219,Z 682.763,A -85,B 0,C 180,E1 -13676.509,E2 -13676.509} C_VEL
LIN {X 0,Y 346.137,Z 684.495,A -85,B 0,C 180,E1 -13677.673,E2 -13677.673} C_VEL
LIN {X 0,Y 346.114,Z 685.802,A -85,B 0,C 180,E1 -13678.836,E2 -13678.836} C_VEL
LIN {X 0,Y 346.145,Z 686.617,A -85,B 0,C 180,E1 -13680,E2 -13680} C_VEL
LIN {X 0,Y 346.177,Z 687.011,A -85,B 0,C 180,E1 -13681.163,E2 -13681.163} C_VEL
LIN {X 0,Y 346.228,Z 686.982,A -85,B 0,C 180,E1 -13682.327,E2 -13682.327} C_VEL
LIN {X 0,Y 346.286,Z 686.474,A -85,B 0,C 180,E1 -13683.491,E2 -13683.491} C_VEL
LIN {X 0,Y 346.448,Z 685.55,A -85,B 0,C 180,E1 -13684.654,E2 -13684.654} C_VEL
LIN {X 0,Y 346.744,Z 684.198,A -85,B 0,C 180,E1 -13685.816,E2 -13685.816} C_VEL
LIN {X 0,Y 347.066,Z 681.296,A -85,B 0,C 180,E1 -13687.563,E2 -13687.563} C_VEL
LIN {X 0,Y 347.652,Z 677.282,A -85,B 0,C 180,E1 -13689.307,E2 -13689.307} C_VEL
LIN {X 0,Y 348.603,Z 671.064,A -85,B 0,C 180,E1 -13691.336,E2 -13691.336} C_VEL
LIN {X 0,Y 349.714,Z 664.27,A -85,B 0,C 180,E1 -13693.067,E2 -13693.067} C_VEL
LIN {X 0,Y 350.993,Z 655.805,A -85,B 0,C 180,E1 -13694.791,E2 -13694.791} C_VEL
LIN {X 0,Y 352.469,Z 646.146,A -85,B 0,C 180,E1 -13696.363,E2 -13696.363} C_VEL
LIN {X 0,Y 353.946,Z 635.474,A -85,B 0,C 180,E1 -13697.76,E2 -13697.76} C_VEL
LIN {X 0,Y 355.329,Z 624.748,A -85,B 0,C 180,E1 -13698.898,E2 -13698.898} C_VEL
LIN {X 0,Y 356.595,Z 613.229,A -85,B 0,C 180,E1 -13699.875,E2 -13699.875} C_VEL
LIN {X 0,Y 357.774,Z 600.523,A -85,B 0,C 180,E1 -13700.707,E2 -13700.707} C_VEL
LIN {X 0,Y 358.8,Z 587.43,A -85,B 0,C 180,E1 -13701.321,E2 -13701.321} C_VEL
LIN {X 0,Y 363.842,Z 502.687,A -85,B 0,C 180,E1 -13703.998,E2 -13703.998} C_VEL
LIN {X 0,Y 361.429,Z 488.948,A -85,B 0,C 180,E1 -13704.888,E2 -13704.888} C_VEL
LIN {X 0,Y 358.372,Z 476.053,A -85,B 0,C 180,E1 -13705.898,E2 -13705.898} C_VEL
LIN {X 0,Y 359.373,Z 468.074,A -85,B 0,C 180,E1 -13707.512,E2 -13707.512} C_VEL
LIN {X 0,Y 358.904,Z 463.304,A -85,B 0,C 180,E1 -13708.669,E2 -13708.669} C_VEL
LIN {X 0,Y 357.289,Z 455.735,A -85,B 0,C 180,E1 -13710.759,E2 -13710.759} C_VEL
LIN {X 0,Y 355.242,Z 448.552,A -85,B 0,C 180,E1 -13713.013,E2 -13713.013} C_VEL
LIN {X 0,Y 353.748,Z 444.05,A -85,B 0,C 180,E1 -13714.589,E2 -13714.589} C_VEL
LIN {X 0,Y 351.515,Z 438.437,A -85,B 0,C 180,E1 -13716.894,E2 -13716.894} C_VEL
LIN {X 0,Y 349.405,Z 433.845,A -85,B 0,C 180,E1 -13719.252,E2 -13719.252} C_VEL
LIN {X 0,Y 348.026,Z 431.407,A -85,B 0,C 180,E1 -13720.887,E2 -13720.887} C_VEL
LIN {X 0,Y 347.758,Z 430.164,A -85,B 0,C 180,E1 -13721.665,E2 -13721.665} C_VEL
LIN {X 0,Y 347.708,Z 430.17,A -85,B 0,C 180,E1 -13725.027,E2 -13725.027} C_VEL
LIN {X 0,Y 347.752,Z 430.166,A -85,B 0,C 180,E1 -13728.397,E2 -13728.397} C_VEL
LIN {X 0,Y 347.775,Z 430.163,A -85,B 0,C 180,E1 -13732.011,E2 -13732.011} C_VEL
LIN {X 0,Y 347.755,Z 430.181,A -85,B 0,C 180,E1 -13733.275,E2 -13733.275} C_VEL
LIN {X 0,Y 348.787,Z 433.039,A -85,B 0,C 180,E1 -13734.737,E2 -13734.737} C_VEL
LIN {X 0,Y 350.3,Z 434.726,A -85,B 0,C 180,E1 -13735.822,E2 -13735.822} C_VEL
LIN {X 0,Y 352.199,Z 438.879,A -85,B 0,C 180,E1 -13737.4,E2 -13737.4} C_VEL
LIN {X 0,Y 354.009,Z 448.681,A -85,B 0,C 180,E1 -13739.588,E2 -13739.588} C_VEL
LIN {X 0,Y 356.206,Z 457.998,A -85,B 0,C 180,E1 -13741.349,E2 -13741.349} C_VEL
LIN {X 0,Y 356.622,Z 469.311,A -85,B 0,C 180,E1 -13742.729,E2 -13742.729} C_VEL
LIN {X 0,Y 357.428,Z 483.867,A -85,B 0,C 180,E1 -13744.27,E2 -13744.27} C_VEL
LIN {X 0,Y 359.949,Z 501.354,A -85,B 0,C 180,E1 -13745.411,E2 -13745.411} C_VEL
LIN {X 0,Y 361.086,Z 514.29,A -85,B 0,C 180,E1 -13746.1,E2 -13746.1} C_VEL
LIN {X 0,Y 361.687,Z 528.257,A -85,B 0,C 180,E1 -13746.75,E2 -13746.75} C_VEL
LIN {X 0,Y 356.804,Z 608.602,A -85,B 0,C 180,E1 -13749.347,E2 -13749.347} C_VEL
LIN {X 0,Y 355.714,Z 621.574,A -85,B 0,C 180,E1 -13749.998,E2 -13749.998} C_VEL
LIN {X 0,Y 354.411,Z 634.633,A -85,B 0,C 180,E1 -13750.901,E2 -13750.901} C_VEL
LIN {X 0,Y 352.912,Z 646.929,A -85,B 0,C 180,E1 -13752.021,E2 -13752.021} C_VEL
LIN {X 0,Y 351.556,Z 658.057,A -85,B 0,C 180,E1 -13753.299,E2 -13753.299} C_VEL
LIN {X 0,Y 350.12,Z 668.929,A -85,B 0,C 180,E1 -13754.873,E2 -13754.873} C_VEL
LIN {X 0,Y 349.038,Z 677.006,A -85,B 0,C 180,E1 -13756.315,E2 -13756.315} C_VEL
LIN {X 0,Y 347.996,Z 684.883,A -85,B 0,C 180,E1 -13758.053,E2 -13758.053} C_VEL
LIN {X 0,Y 347.372,Z 690.278,A -85,B 0,C 180,E1 -13759.509,E2 -13759.509} C_VEL
LIN {X 0,Y 346.778,Z 695.484,A -85,B 0,C 180,E1 -13761.257,E2 -13761.257} C_VEL
LIN {X 0,Y 346.423,Z 699.472,A -85,B 0,C 180,E1 -13763.008,E2 -13763.008} C_VEL
LIN {X 0,Y 346.289,Z 701.528,A -85,B 0,C 180,E1 -13764.176,E2 -13764.176} C_VEL
LIN {X 0,Y 346.256,Z 703.078,A -85,B 0,C 180,E1 -13765.343,E2 -13765.343} C_VEL
LIN {X 0,Y 346.205,Z 704.181,A -85,B 0,C 180,E1 -13766.508,E2 -13766.508} C_VEL
LIN {X 0,Y 346.144,Z 704.851,A -85,B 0,C 180,E1 -13767.673,E2 -13767.673} C_VEL
LIN {X 0,Y 346.238,Z 705.259,A -85,B 0,C 180,E1 -13770,E2 -13770} C_VEL
LIN {X 0,Y 346.176,Z 705.034,A -85,B 0,C 180,E1 -13771.163,E2 -13771.163} C_VEL
LIN {X 0,Y 346.206,Z 703.405,A -85,B 0,C 180,E1 -13773.492,E2 -13773.492} C_VEL
LIN {X 0,Y 346.24,Z 701.97,A -85,B 0,C 180,E1 -13774.657,E2 -13774.657} C_VEL
LIN {X 0,Y 346.279,Z 699.723,A -85,B 0,C 180,E1 -13776.015,E2 -13776.015} C_VEL
LIN {X 0,Y 346.577,Z 694.936,A -85,B 0,C 180,E1 -13778.161,E2 -13778.161} C_VEL
LIN {X 0,Y 347.123,Z 688.692,A -85,B 0,C 180,E1 -13780.204,E2 -13780.204} C_VEL
LIN {X 0,Y 347.794,Z 681.88,A -85,B 0,C 180,E1 -13781.954,E2 -13781.954} C_VEL
LIN {X 0,Y 348.641,Z 674.912,A -85,B 0,C 180,E1 -13783.404,E2 -13783.404} C_VEL
LIN {X 0,Y 349.599,Z 666.489,A -85,B 0,C 180,E1 -13784.852,E2 -13784.852} C_VEL
LIN {X 0,Y 350.682,Z 656.061,A -85,B 0,C 180,E1 -13786.294,E2 -13786.294} C_VEL
LIN {X 0,Y 351.792,Z 645.732,A -85,B 0,C 180,E1 -13787.438,E2 -13787.438} C_VEL
LIN {X 0,Y 352.897,Z 634.355,A -85,B 0,C 180,E1 -13788.431,E2 -13788.431} C_VEL
LIN {X 0,Y 353.621,Z 627.118,A -85,B 0,C 180,E1 -13788.993,E2 -13788.993} C_VEL
LIN {X 0,Y 355.45,Z 613.371,A -85,B 0,C 180,E1 -13790.093,E2 -13790.093} C_VEL
LIN {X 0,Y 357.04,Z 599.783,A -85,B 0,C 180,E1 -13790.902,E2 -13790.902} C_VEL
LIN {X 0,Y 358.224,Z 585.897,A -85,B 0,C 180,E1 -13791.508,E2 -13791.508} C_VEL
LIN {X 0,Y 361.474,Z 526.255,A -85,B 0,C 180,E1 -13793.364,E2 -13793.364} C_VEL
LIN {X 0,Y 360.524,Z 510.633,A -85,B 0,C 180,E1 -13794.084,E2 -13794.084} C_VEL
LIN {X 0,Y 358.517,Z 494.552,A -85,B 0,C 180,E1 -13794.989,E2 -13794.989} C_VEL
LIN {X 0,Y 355.659,Z 479.388,A -85,B 0,C 180,E1 -13796.03,E2 -13796.03} C_VEL
LIN {X 0,Y 354.028,Z 471.637,A -85,B 0,C 180,E1 -13796.655,E2 -13796.655} C_VEL
LIN {X 0,Y 355.764,Z 462.061,A -85,B 0,C 180,E1 -13798.892,E2 -13798.892} C_VEL
LIN {X 0,Y 354.968,Z 455.949,A -85,B 0,C 180,E1 -13800.652,E2 -13800.652} C_VEL
LIN {X 0,Y 353.193,Z 447.942,A -85,B 0,C 180,E1 -13803.307,E2 -13803.307} C_VEL
LIN {X 0,Y 351.101,Z 440.278,A -85,B 0,C 180,E1 -13806.337,E2 -13806.337} C_VEL
LIN {X 0,Y 349.62,Z 435.721,A -85,B 0,C 180,E1 -13808.547,E2 -13808.547} C_VEL
LIN {X 0,Y 348.214,Z 431.949,A -85,B 0,C 180,E1 -13810.811,E2 -13810.811} C_VEL
LIN {X 0,Y 347.743,Z 430.168,A -85,B 0,C 180,E1 -13812.124,E2 -13812.124} C_VEL
LIN {X 0,Y 347.707,Z 430.172,A -85,B 0,C 180,E1 -13815.027,E2 -13815.027} C_VEL
LIN {X 0,Y 347.752,Z 430.166,A -85,B 0,C 180,E1 -13818.397,E2 -13818.397} C_VEL
LIN {X 0,Y 347.776,Z 430.165,A -85,B 0,C 180,E1 -13822.011,E2 -13822.011} C_VEL
LIN {X 0,Y 347.746,Z 430.167,A -85,B 0,C 180,E1 -13825.536,E2 -13825.536} C_VEL
LIN {X 0,Y 347.747,Z 430.169,A -85,B 0,C 180,E1 -13828.301,E2 -13828.301} C_VEL
LIN {X 0,Y 347.805,Z 430.352,A -85,B 0,C 180,E1 -13830.33,E2 -13830.33} C_VEL
LIN {X 0,Y 348.793,Z 433.441,A -85,B 0,C 180,E1 -13832.628,E2 -13832.628} C_VEL
LIN {X 0,Y 351.05,Z 436.672,A -85,B 0,C 180,E1 -13833.206,E2 -13833.206} C_VEL
LIN {X 0,Y 352.3,Z 438.438,A -85,B 0,C 180,E1 -13833.519,E2 -13833.519} C_VEL
LIN {X 0,Y 356.636,Z 444.872,A -85,B 0,C 180,E1 -13834.529,E2 -13834.529} C_VEL
LIN {X 0,Y 361.86,Z 454.348,A -85,B 0,C 180,E1 -13835.719,E2 -13835.719} C_VEL
LIN {X 0,Y 364.455,Z 459.735,A -85,B 0,C 180,E1 -13836.3,E2 -13836.3} C_VEL
LIN {X 0,Y 360.131,Z 529.475,A -85,B 0,C 180,E1 -13838.536,E2 -13838.536} C_VEL
LIN {X 0,Y 359.423,Z 542.485,A -85,B 0,C 180,E1 -13839.093,E2 -13839.093} C_VEL
LIN {X 0,Y 358.704,Z 554.213,A -85,B 0,C 180,E1 -13839.799,E2 -13839.799} C_VEL
LIN {X 0,Y 357.503,Z 567.287,A -85,B 0,C 180,E1 -13840.833,E2 -13840.833} C_VEL
LIN {X 0,Y 356.08,Z 579.117,A -85,B 0,C 180,E1 -13842.038,E2 -13842.038} C_VEL
LIN {X 0,Y 354.7,Z 589.03,A -85,B 0,C 180,E1 -13843.304,E2 -13843.304} C_VEL
LIN {X 0,Y 353.446,Z 598.096,A -85,B 0,C 180,E1 -13844.724,E2 -13844.724} C_VEL
LIN {X 0,Y 352.045,Z 606.858,A -85,B 0,C 180,E1 -13846.434,E2 -13846.434} C_VEL
LIN {X 0,Y 350.772,Z 613.901,A -85,B 0,C 180,E1 -13848.149,E2 -13848.149} C_VEL
LIN {X 0,Y 349.791,Z 619.544,A -85,B 0,C 180,E1 -13849.903,E2 -13849.903} C_VEL
LIN {X 0,Y 348.635,Z 624.427,A -85,B 0,C 180,E1 -13851.888,E2 -13851.888} C_VEL
LIN {X 0,Y 348.284,Z 626.563,A -85,B 0,C 180,E1 -13853.046,E2 -13853.046} C_VEL
LIN {X 0,Y 347.949,Z 628.248,A -85,B 0,C 180,E1 -13854.204,E2 -13854.204} C_VEL
LIN {X 0,Y 347.586,Z 629.457,A -85,B 0,C 180,E1 -13855.361,E2 -13855.361} C_VEL
LIN {X 0,Y 347.216,Z 630.259,A -85,B 0,C 180,E1 -13856.519,E2 -13856.519} C_VEL
LIN {X 0,Y 346.943,Z 630.641,A -85,B 0,C 180,E1 -13857.678,E2 -13857.678} C_VEL
LIN {X 0,Y 346.794,Z 630.547,A -85,B 0,C 180,E1 -13858.839,E2 -13858.839} C_VEL
LIN {X 0,Y 346.74,Z 630.026,A -85,B 0,C 180,E1 -13860,E2 -13860} C_VEL
LIN {X 0,Y 346.775,Z 629.094,A -85,B 0,C 180,E1 -13861.161,E2 -13861.161} C_VEL
LIN {X 0,Y 346.812,Z 627.716,A -85,B 0,C 180,E1 -13862.323,E2 -13862.323} C_VEL
LIN {X 0,Y 347.051,Z 624.793,A -85,B 0,C 180,E1 -13864.064,E2 -13864.064} C_VEL
LIN {X 0,Y 347.152,Z 620.799,A -85,B 0,C 180,E1 -13865.81,E2 -13865.81} C_VEL
LIN {X 0,Y 347.469,Z 615.274,A -85,B 0,C 180,E1 -13867.653,E2 -13867.653} C_VEL
LIN {X 0,Y 347.878,Z 607.848,A -85,B 0,C 180,E1 -13869.594,E2 -13869.594} C_VEL
LIN {X 0,Y 348.515,Z 599.372,A -85,B 0,C 180,E1 -13871.339,E2 -13871.339} C_VEL
LIN {X 0,Y 349.085,Z 590.74,A -85,B 0,C 180,E1 -13872.795,E2 -13872.795} C_VEL
LIN {X 0,Y 349.86,Z 580.205,A -85,B 0,C 180,E1 -13874.246,E2 -13874.246} C_VEL
LIN {X 0,Y 350.573,Z 569.081,A -85,B 0,C 180,E1 -13875.479,E2 -13875.479} C_VEL
LIN {X 0,Y 351.173,Z 556.808,A -85,B 0,C 180,E1 -13876.57,E2 -13876.57} C_VEL
LIN {X 0,Y 351.738,Z 543.917,A -85,B 0,C 180,E1 -13877.44,E2 -13877.44} C_VEL
LIN {X 0,Y 352.183,Z 530.77,A -85,B 0,C 180,E1 -13878.093,E2 -13878.093} C_VEL
LIN {X 0,Y 352.53,Z 514.685,A -85,B 0,C 180,E1 -13878.601,E2 -13878.601} C_VEL
LIN {X 0,Y 354.209,Z 449.877,A -85,B 0,C 180,E1 -13880.344,E2 -13880.344} C_VEL
LIN {X 0,Y 347.816,Z 430.165,A -85,B 0,C 180,E1 -13881.19,E2 -13881.19} C_VEL
LIN {X 0,Y 347.814,Z 430.159,A -85,B 0,C 180,E1 -13885.108,E2 -13885.108} C_VEL
LIN {X 0,Y 347.81,Z 430.154,A -85,B 0,C 180,E1 -13887.694,E2 -13887.694} C_VEL
LIN {X 0,Y 347.751,Z 430.166,A -85,B 0,C 180,E1 -13890.348,E2 -13890.348} C_VEL
LIN {X 0,Y 347.75,Z 430.144,A -85,B 0,C 180,E1 -13894.044,E2 -13894.044} C_VEL
LIN {X 0,Y 347.764,Z 430.17,A -85,B 0,C 180,E1 -13897.321,E2 -13897.321} C_VEL
LIN {X 0,Y 347.734,Z 430.154,A -85,B 0,C 180,E1 -13900.297,E2 -13900.297} C_VEL
LIN {X 0,Y 347.725,Z 430.174,A -85,B 0,C 180,E1 -13903.408,E2 -13903.408} C_VEL
LIN {X 0,Y 347.727,Z 430.161,A -85,B 0,C 180,E1 -13906.686,E2 -13906.686} C_VEL
LIN {X 0,Y 347.749,Z 430.159,A -85,B 0,C 180,E1 -13910.173,E2 -13910.173} C_VEL
LIN {X 0,Y 347.763,Z 430.162,A -85,B 0,C 180,E1 -13912.679,E2 -13912.679} C_VEL
LIN {X 0,Y 347.75,Z 430.164,A -85,B 0,C 180,E1 -13915.956,E2 -13915.956} C_VEL
LIN {X 0,Y 347.783,Z 430.357,A -85,B 0,C 180,E1 -13918.559,E2 -13918.559} C_VEL
LIN {X 0,Y 350.768,Z 442.333,A -85,B 0,C 180,E1 -13921.258,E2 -13921.258} C_VEL
LIN {X 0,Y 353.3,Z 454.535,A -85,B 0,C 180,E1 -13923.867,E2 -13923.867} C_VEL
LIN {X 0,Y 353.018,Z 462.147,A -85,B 0,C 180,E1 -13925.287,E2 -13925.287} C_VEL
LIN {X 0,Y 352.506,Z 473.039,A -85,B 0,C 180,E1 -13927.197,E2 -13927.197} C_VEL
LIN {X 0,Y 357.236,Z 500.003,A -85,B 0,C 180,E1 -13928.094,E2 -13928.094} C_VEL
LIN {X 0,Y 355.701,Z 582.324,A -85,B 0,C 180,E1 -13929.771,E2 -13929.771} C_VEL
LIN {X 0,Y 355.232,Z 595.378,A -85,B 0,C 180,E1 -13930.233,E2 -13930.233} C_VEL
LIN {X 0,Y 354.493,Z 606.776,A -85,B 0,C 180,E1 -13930.831,E2 -13930.831} C_VEL
LIN {X 0,Y 353.476,Z 619.458,A -85,B 0,C 180,E1 -13931.751,E2 -13931.751} C_VEL
LIN {X 0,Y 352.281,Z 631.673,A -85,B 0,C 180,E1 -13932.916,E2 -13932.916} C_VEL
LIN {X 0,Y 351.378,Z 641.935,A -85,B 0,C 180,E1 -13934.186,E2 -13934.186} C_VEL
LIN {X 0,Y 350.06,Z 652.289,A -85,B 0,C 180,E1 -13935.763,E2 -13935.763} C_VEL
LIN {X 0,Y 348.996,Z 659.935,A -85,B 0,C 180,E1 -13937.202,E2 -13937.202} C_VEL
LIN {X 0,Y 348.134,Z 667.38,A -85,B 0,C 180,E1 -13938.943,E2 -13938.943} C_VEL
LIN {X 0,Y 347.374,Z 673.354,A -85,B 0,C 180,E1 -13940.685,E2 -13940.685} C_VEL
LIN {X 0,Y 346.891,Z 678.078,A -85,B 0,C 180,E1 -13942.433,E2 -13942.433} C_VEL
LIN {X 0,Y 346.571,Z 681.691,A -85,B 0,C 180,E1 -13944.181,E2 -13944.181} C_VEL
LIN {X 0,Y 346.423,Z 683.551,A -85,B 0,C 180,E1 -13945.345,E2 -13945.345} C_VEL
LIN {X 0,Y 346.248,Z 684.973,A -85,B 0,C 180,E1 -13946.509,E2 -13946.509} C_VEL
LIN {X 0,Y 346.154,Z 686.582,A -85,B 0,C 180,E1 -13948.837,E2 -13948.837} C_VEL
LIN {X 0,Y 346.151,Z 686.816,A -85,B 0,C 180,E1 -13950,E2 -13950} C_VEL
LIN {X 0,Y 346.154,Z 686.624,A -85,B 0,C 180,E1 -13951.163,E2 -13951.163} C_VEL
LIN {X 0,Y 346.247,Z 685.069,A -85,B 0,C 180,E1 -13953.491,E2 -13953.491} C_VEL
LIN {X 0,Y 346.421,Z 683.701,A -85,B 0,C 180,E1 -13954.655,E2 -13954.655} C_VEL
LIN {X 0,Y 346.715,Z 680.291,A -85,B 0,C 180,E1 -13956.663,E2 -13956.663} C_VEL
LIN {X 0,Y 347.172,Z 675.352,A -85,B 0,C 180,E1 -13958.733,E2 -13958.733} C_VEL
LIN {X 0,Y 347.867,Z 669.891,A -85,B 0,C 180,E1 -13960.476,E2 -13960.476} C_VEL
LIN {X 0,Y 348.752,Z 663.043,A -85,B 0,C 180,E1 -13962.216,E2 -13962.216} C_VEL
LIN {X 0,Y 349.772,Z 654.478,A -85,B 0,C 180,E1 -13963.953,E2 -13963.953} C_VEL
LIN {X 0,Y 350.914,Z 645.84,A -85,B 0,C 180,E1 -13965.366,E2 -13965.366} C_VEL
LIN {X 0,Y 351.076,Z 644.469,A -85,B 0,C 180,E1 -13965.566,E2 -13965.566} C_VEL
LIN {X 0,Y 350.744,Z 641.561,A -85,B 0,C 180,E1 -13966.011,E2 -13966.011} C_VEL
LIN {X 0,Y 348.425,Z 637.029,A -85,B 0,C 180,E1 -13966.744,E2 -13966.744} C_VEL
LIN {X 0,Y 346.141,Z 632.315,A -85,B 0,C 180,E1 -13967.444,E2 -13967.444} C_VEL
LIN {X 0,Y 345.852,Z 629.069,A -85,B 0,C 180,E1 -13967.828,E2 -13967.828} C_VEL
LIN {X 0,Y 346.995,Z 617.409,A -85,B 0,C 180,E1 -13968.909,E2 -13968.909} C_VEL
LIN {X 0,Y 348.036,Z 604.97,A -85,B 0,C 180,E1 -13969.77,E2 -13969.77} C_VEL
LIN {X 0,Y 348.687,Z 591.976,A -85,B 0,C 180,E1 -13970.423,E2 -13970.423} C_VEL
LIN {X 0,Y 349.187,Z 579.272,A -85,B 0,C 180,E1 -13970.816,E2 -13970.816} C_VEL
LIN {X 0,Y 350.679,Z 500.948,A -85,B 0,C 180,E1 -13972.426,E2 -13972.426} C_VEL
LIN {X 0,Y 346.399,Z 476.425,A -85,B 0,C 180,E1 -13973.263,E2 -13973.263} C_VEL
LIN {X 0,Y 345.743,Z 472.888,A -85,B 0,C 180,E1 -13973.405,E2 -13973.405} C_VEL
LIN {X 0,Y 346.639,Z 457.74,A -85,B 0,C 180,E1 -13976.166,E2 -13976.166} C_VEL
LIN {X 0,Y 344.89,Z 448.307,A -85,B 0,C 180,E1 -13978.156,E2 -13978.156} C_VEL
LIN {X 0,Y 342.031,Z 436.05,A -85,B 0,C 180,E1 -13980.91,E2 -13980.91} C_VEL
LIN {X 0,Y 340.705,Z 431.051,A -85,B 0,C 180,E1 -13982.084,E2 -13982.084} C_VEL
LIN {X 0,Y 340.72,Z 431.045,A -85,B 0,C 180,E1 -13985.279,E2 -13985.279} C_VEL
LIN {X 0,Y 340.712,Z 431.044,A -85,B 0,C 180,E1 -13988.386,E2 -13988.386} C_VEL
LIN {X 0,Y 340.701,Z 431.047,A -85,B 0,C 180,E1 -13992.045,E2 -13992.045} C_VEL
LIN {X 0,Y 340.687,Z 431.052,A -85,B 0,C 180,E1 -13995.462,E2 -13995.462} C_VEL
LIN {X 0,Y 340.688,Z 431.038,A -85,B 0,C 180,E1 -13998.69,E2 -13998.69} C_VEL
